# B&R Automation Studio project MotionTestBenchMaster (part 32)

```iecst
                               VAR_RNS_SEQ.Device.FSB201.ALR := FALSE;                                                 (* STEP: 93 FSB201*)
                               VAR_RNS_SEQ.Device.FSB201.WAIT_OFF := FALSE;
                               VAR_RNS_SEQ.Device.FSB201.WAIT_ON := FALSE;

                               VAR_RNS_SEQ.Device.FTB201.ALR_HighLimitEn := FALSE;                                     (* STEP: 93 FTB201*)
                               VAR_RNS_SEQ.Device.FTB201.ALR_HighLimitSP := 0;
                               VAR_RNS_SEQ.Device.FTB201.ALR_LowLimitEn := FALSE;
                               VAR_RNS_SEQ.Device.FTB201.ALR_LowLimitSP := 0;
                               VAR_RNS_SEQ.Device.FTB201.SP := 0;
                               VAR_RNS_SEQ.Device.FTB201.CMP := 0;
                               VAR_RNS_SEQ.Device.FTB201.MinDev := 0;
                               VAR_RNS_SEQ.Device.FTB201.MaxDev := 0;

                               VAR_RNS_SEQ.Device.FTB202.ALR_HighLimitEn := FALSE;                                     (* STEP: 93 FTB202*)
                               VAR_RNS_SEQ.Device.FTB202.ALR_HighLimitSP := 0;
                               VAR_RNS_SEQ.Device.FTB202.ALR_LowLimitEn := FALSE;
                               VAR_RNS_SEQ.Device.FTB202.ALR_LowLimitSP := 0;
                               VAR_RNS_SEQ.Device.FTB202.SP := 0;
                               VAR_RNS_SEQ.Device.FTB202.CMP := 0;
                               VAR_RNS_SEQ.Device.FTB202.MinDev := 0;
                               VAR_RNS_SEQ.Device.FTB202.MaxDev := 0;

                               VAR_RNS_SEQ.Device.PTB220.ALR_HighLimitEn := FALSE;                                     (* STEP: 93 PTB220*)
                               VAR_RNS_SEQ.Device.PTB220.ALR_HighLimitSP := 0;
                               VAR_RNS_SEQ.Device.PTB220.ALR_LowLimitEn := FALSE;
                               VAR_RNS_SEQ.Device.PTB220.ALR_LowLimitSP := 0;
                               VAR_RNS_SEQ.Device.PTB220.SP := 0;
                               VAR_RNS_SEQ.Device.PTB220.CMP := 0;
                               VAR_RNS_SEQ.Device.PTB220.MinDev := 0;
                               VAR_RNS_SEQ.Device.PTB220.MaxDev := 0;

                               VAR_RNS_SEQ.Device.PTB270.ALR_HighLimitEn := FALSE;                                     (* STEP: 93 PTB270*)
                               VAR_RNS_SEQ.Device.PTB270.ALR_HighLimitSP := 0;
                               VAR_RNS_SEQ.Device.PTB270.ALR_LowLimitEn := FALSE;
                               VAR_RNS_SEQ.Device.PTB270.ALR_LowLimitSP := 0;
                               VAR_RNS_SEQ.Device.PTB270.SP := 0;
                               VAR_RNS_SEQ.Device.PTB270.CMP := 0;
                               VAR_RNS_SEQ.Device.PTB270.MinDev := 0;
                               VAR_RNS_SEQ.Device.PTB270.MaxDev := 0;

                               VAR_RNS_SEQ.Device.LTB202.ALR_HighLimitEn := FALSE;                                     (* STEP: 93 LTB202*)
                               VAR_RNS_SEQ.Device.LTB202.ALR_HighLimitSP := 0;
                               VAR_RNS_SEQ.Device.LTB202.ALR_LowLimitEn := FALSE;
                               VAR_RNS_SEQ.Device.LTB202.ALR_LowLimitSP := 0;
                               VAR_RNS_SEQ.Device.LTB202.SP := 0;
                               VAR_RNS_SEQ.Device.LTB202.CMP := 0;
                               VAR_RNS_SEQ.Device.LTB202.MinDev := 0;
                               VAR_RNS_SEQ.Device.LTB202.MaxDev := 0;

                               VAR_RNS_SEQ.Device.PTB290.ALR_HighLimitEn := FALSE;                                     (* STEP: 93 PTB290*)
                               VAR_RNS_SEQ.Device.PTB290.ALR_HighLimitSP := 0;
                               VAR_RNS_SEQ.Device.PTB290.ALR_LowLimitEn := FALSE;
                               VAR_RNS_SEQ.Device.PTB290.ALR_LowLimitSP := 0;
                               VAR_RNS_SEQ.Device.PTB290.SP := 0;
                               VAR_RNS_SEQ.Device.PTB290.CMP := 0;
                               VAR_RNS_SEQ.Device.PTB290.MinDev := 0;
                               VAR_RNS_SEQ.Device.PTB290.MaxDev := 0;

                               VAR_RNS_SEQ.Mem.ContainersStop := TRUE;                                                 (* STEP: 93 *)
                               VAR_RNS_SEQ.Mem.ControlInsercion := FALSE;                                              (* STEP: 93 *)
                               VAR_RNS_SEQ.Mem.ControlContinous := FALSE;                                              (* STEP: 93 *)
                               VAR_RNS_SEQ.Mem.PBAbortEnable := TRUE;                                                  (* STEP: 93 PB Abort Sequence Enable*)
                               VAR_RNS_SEQ.Mem.PBStopEnable := TRUE;                                                   (* STEP: 93 PB Stop Sequence Enable*)
                               VAR_RNS_SEQ.Mem.PBStartEnable := FALSE;                                                 (* STEP: 93 PB Start Sequence Enable*)
                               VAR_RNS_SEQ.Mem.ByPassed := TRUE;                                                       (* STEP: 93 *)
                               VAR_RNS_SEQ.Mem.InsercionDevice := FALSE;                                               (* STEP: 93 *)
                               VAR_RNS_SEQ.Mem.AirTreatmentControl := FALSE;                                           (* STEP: 93 *)
                               VAR_RNS_SEQ.Mem.WaterTreatmentControl := FALSE;                                         (* STEP: 93 *)
                               VAR_RNS_SEQ.Mem.SpeedReductionControl := FALSE;                                         (* STEP: 93 *)
                               VAR_RNS_SEQ.Mem.ByPassRequest := FALSE;                                                 (* STEP: 93 *)
                               VAR_RNS_SEQ.Mem.CopAfterCipRequest := FALSE;                                            (* STEP: 93 *)
                               VAR_RNS_SEQ.Mem.NoBoNoSprayInsercion := FALSE;                                          (* STEP: 93 *)

                               VAR_RNS_SEQ.ITC.WTT_ProductRequest := FALSE;                                            (* STEP: 93 *)
                               VAR_RNS_SEQ.ITC.WTT_ProductionRunning := FALSE;                                         (* STEP: 93 *)

                       94: (* BYPASSED - Rinser Inserted  *)

                               VAR_RNS_SEQ.Device.AVB224.AutoCnd := FALSE;                                             (* STEP: 94 AVB224*)
                               VAR_RNS_SEQ.Device.AVB224.EnableCnd := FALSE;
                               VAR_RNS_SEQ.Device.AVB228.AutoCnd := FALSE;                                             (* STEP: 94 AVB228*)
                               VAR_RNS_SEQ.Device.AVB228.EnableCnd := FALSE;
                               VAR_RNS_SEQ.Device.AVB234.AutoCnd := FALSE;                                             (* STEP: 94 AVB234*)
                               VAR_RNS_SEQ.Device.AVB234.EnableCnd := FALSE;
                               VAR_RNS_SEQ.Device.AVB261.AutoCnd := FALSE;                                             (* STEP: 94 AVB261*)
                               VAR_RNS_SEQ.Device.AVB261.EnableCnd := FALSE;
                               VAR_RNS_SEQ.Device.AVB264.AutoCnd := FALSE;                                             (* STEP: 94 AVB264*)
                               VAR_RNS_SEQ.Device.AVB264.EnableCnd := FALSE;
                               VAR_RNS_SEQ.Device.AVB265.AutoCnd := FALSE;                                             (* STEP: 94 AVB265*)
                               VAR_RNS_SEQ.Device.AVB265.EnableCnd := FALSE;
                               VAR_RNS_SEQ.Device.AVB266.AutoCnd := FALSE;                                             (* STEP: 94 AVB266*)
                               VAR_RNS_SEQ.Device.AVB266.EnableCnd := FALSE;
                               VAR_RNS_SEQ.Device.AVB267.AutoCnd := FALSE;                                             (* STEP: 94 AVB267*)
                               VAR_RNS_SEQ.Device.AVB267.EnableCnd := FALSE;
                               VAR_RNS_SEQ.Device.AVB268.AutoCnd := FALSE;                                             (* STEP: 94 AVB268*)
                               VAR_RNS_SEQ.Device.AVB268.EnableCnd := FALSE;
                               VAR_RNS_SEQ.Device.AVB273.AutoCnd := FALSE;                                             (* STEP: 94 AVB273*)
                               VAR_RNS_SEQ.Device.AVB273.EnableCnd := FALSE;
                               VAR_RNS_SEQ.Device.AVB294.AutoCnd := FALSE;                                             (* STEP: 94 AVB294*)
                               VAR_RNS_SEQ.Device.AVB294.EnableCnd := FALSE;

                               VAR_RNS_SEQ.Device.PPB209_PID.PID_Enable := FALSE;                                      (* STEP: 94 PPB209*)
                               VAR_RNS_SEQ.Device.PPB209_PID.PID_Mode := FALSE;
                               VAR_RNS_SEQ.Device.PPB209_PID.Auto_SP_Value := 0;
                               VAR_RNS_SEQ.Device.PPB209_PID.FIX_Value := 0;

                               VAR_RNS_SEQ.Device.RVB202_PID.PID_Enable := FALSE;                                      (* STEP: 94 *)
                               VAR_RNS_SEQ.Device.RVB202_PID.PID_Mode := FALSE;
                               VAR_RNS_SEQ.Device.RVB202_PID.Auto_SP_Value := 0;
                               VAR_RNS_SEQ.Device.RVB202_PID.FIX_Value := 0;

                               VAR_RNS_SEQ.Device.FSB220.ALR := FALSE;                                                 (* STEP: 94 FSB220*)
                               VAR_RNS_SEQ.Device.FSB220.WAIT_OFF := FALSE;
                               VAR_RNS_SEQ.Device.FSB220.WAIT_ON := FALSE;

                               VAR_RNS_SEQ.Device.LSB209.ALR := FALSE;                                                 (* STEP: 94 LSB209*)
                               VAR_RNS_SEQ.Device.LSB209.WAIT_OFF := FALSE;
                               VAR_RNS_SEQ.Device.LSB209.WAIT_ON := FALSE;

                               VAR_RNS_SEQ.Device.LSB210.ALR := FALSE;                                                 (* STEP: 94 LSB210*)
                               VAR_RNS_SEQ.Device.LSB210.WAIT_OFF := FALSE;
                               VAR_RNS_SEQ.Device.LSB210.WAIT_ON := FALSE;

                               VAR_RNS_SEQ.Device.LSB299.ALR := FALSE;                                                 (* STEP: 94 *)
                               VAR_RNS_SEQ.Device.LSB299.WAIT_OFF := FALSE;
                               VAR_RNS_SEQ.Device.LSB299.WAIT_ON := FALSE;

                               VAR_RNS_SEQ.Device.FSB201.ALR := FALSE;                                                 (* STEP: 94 FSB201*)
                               VAR_RNS_SEQ.Device.FSB201.WAIT_OFF := FALSE;
                               VAR_RNS_SEQ.Device.FSB201.WAIT_ON := FALSE;

                               VAR_RNS_SEQ.Device.FTB201.ALR_HighLimitEn := FALSE;                                     (* STEP: 94 FTB201*)
                               VAR_RNS_SEQ.Device.FTB201.ALR_HighLimitSP := 0;
                               VAR_RNS_SEQ.Device.FTB201.ALR_LowLimitEn := FALSE;
                               VAR_RNS_SEQ.Device.FTB201.ALR_LowLimitSP := 0;
                               VAR_RNS_SEQ.Device.FTB201.SP := 0;
                               VAR_RNS_SEQ.Device.FTB201.CMP := 0;
                               VAR_RNS_SEQ.Device.FTB201.MinDev := 0;
                               VAR_RNS_SEQ.Device.FTB201.MaxDev := 0;

                               VAR_RNS_SEQ.Device.FTB202.ALR_HighLimitEn := FALSE;                                     (* STEP: 94 FTB202*)
                               VAR_RNS_SEQ.Device.FTB202.ALR_HighLimitSP := 0;
                               VAR_RNS_SEQ.Device.FTB202.ALR_LowLimitEn := FALSE;
                               VAR_RNS_SEQ.Device.FTB202.ALR_LowLimitSP := 0;
                               VAR_RNS_SEQ.Device.FTB202.SP := 0;
                               VAR_RNS_SEQ.Device.FTB202.CMP := 0;
                               VAR_RNS_SEQ.Device.FTB202.MinDev := 0;
                               VAR_RNS_SEQ.Device.FTB202.MaxDev := 0;

                               VAR_RNS_SEQ.Device.PTB220.ALR_HighLimitEn := FALSE;                                     (* STEP: 94 PTB220*)
                               VAR_RNS_SEQ.Device.PTB220.ALR_HighLimitSP := 0;
                               VAR_RNS_SEQ.Device.PTB220.ALR_LowLimitEn := FALSE;
                               VAR_RNS_SEQ.Device.PTB220.ALR_LowLimitSP := 0;
                               VAR_RNS_SEQ.Device.PTB220.SP := 0;
                               VAR_RNS_SEQ.Device.PTB220.CMP := 0;
                               VAR_RNS_SEQ.Device.PTB220.MinDev := 0;
                               VAR_RNS_SEQ.Device.PTB220.MaxDev := 0;

                               VAR_RNS_SEQ.Device.PTB270.ALR_HighLimitEn := FALSE;                                     (* STEP: 94 PTB270*)
                               VAR_RNS_SEQ.Device.PTB270.ALR_HighLimitSP := 0;
                               VAR_RNS_SEQ.Device.PTB270.ALR_LowLimitEn := FALSE;
                               VAR_RNS_SEQ.Device.PTB270.ALR_LowLimitSP := 0;
                               VAR_RNS_SEQ.Device.PTB270.SP := 0;
                               VAR_RNS_SEQ.Device.PTB270.CMP := 0;
                               VAR_RNS_SEQ.Device.PTB270.MinDev := 0;
                               VAR_RNS_SEQ.Device.PTB270.MaxDev := 0;

                               VAR_RNS_SEQ.Device.LTB202.ALR_HighLimitEn := FALSE;                                     (* STEP: 94 LTB202*)
                               VAR_RNS_SEQ.Device.LTB202.ALR_HighLimitSP := 0;
                               VAR_RNS_SEQ.Device.LTB202.ALR_LowLimitEn := FALSE;
                               VAR_RNS_SEQ.Device.LTB202.ALR_LowLimitSP := 0;
                               VAR_RNS_SEQ.Device.LTB202.SP := 0;
                               VAR_RNS_SEQ.Device.LTB202.CMP := 0;
                               VAR_RNS_SEQ.Device.LTB202.MinDev := 0;
                               VAR_RNS_SEQ.Device.LTB202.MaxDev := 0;

                               VAR_RNS_SEQ.Device.PTB290.ALR_HighLimitEn := FALSE;                                     (* STEP: 94 PTB290*)
                               VAR_RNS_SEQ.Device.PTB290.ALR_HighLimitSP := 0;
                               VAR_RNS_SEQ.Device.PTB290.ALR_LowLimitEn := FALSE;
                               VAR_RNS_SEQ.Device.PTB290.ALR_LowLimitSP := 0;
                               VAR_RNS_SEQ.Device.PTB290.SP := 0;
                               VAR_RNS_SEQ.Device.PTB290.CMP := 0;
                               VAR_RNS_SEQ.Device.PTB290.MinDev := 0;
                               VAR_RNS_SEQ.Device.PTB290.MaxDev := 0;

                               VAR_RNS_SEQ.Mem.ContainersStop := TRUE;                                                 (* STEP: 94 *)
                               VAR_RNS_SEQ.Mem.ControlInsercion := FALSE;                                              (* STEP: 94 *)
                               VAR_RNS_SEQ.Mem.ControlContinous := FALSE;                                              (* STEP: 94 *)
                               VAR_RNS_SEQ.Mem.PBAbortEnable := TRUE;                                                  (* STEP: 94 PB Abort Sequence Enable*)
                               VAR_RNS_SEQ.Mem.PBStopEnable := TRUE;                                                   (* STEP: 94 PB Stop Sequence Enable*)
                               VAR_RNS_SEQ.Mem.PBStartEnable := FALSE;                                                 (* STEP: 94 PB Start Sequence Enable*)
                               VAR_RNS_SEQ.Mem.ByPassed := FALSE;                                                      (* STEP: 94 *)
                               VAR_RNS_SEQ.Mem.InsercionDevice := FALSE;                                               (* STEP: 94 *)
                               VAR_RNS_SEQ.Mem.AirTreatmentControl := FALSE;                                           (* STEP: 94 *)
                               VAR_RNS_SEQ.Mem.WaterTreatmentControl := FALSE;                                         (* STEP: 94 *)
                               VAR_RNS_SEQ.Mem.SpeedReductionControl := FALSE;                                         (* STEP: 94 *)
                               VAR_RNS_SEQ.Mem.ByPassRequest := TRUE;                                                  (* STEP: 94 *)
                               VAR_RNS_SEQ.Mem.CopAfterCipRequest := FALSE;                                            (* STEP: 94 *)
                               VAR_RNS_SEQ.Mem.NoBoNoSprayInsercion := FALSE;                                          (* STEP: 94 *)

                               VAR_RNS_SEQ.ITC.WTT_ProductRequest := FALSE;                                            (* STEP: 94 *)
                               VAR_RNS_SEQ.ITC.WTT_ProductionRunning := FALSE;                                         (* STEP: 94 *)

                       95..100: (* Spare Steps *)

               ELSE
                               RNS_StepStop;
               END_CASE
END_ACTION
```

#### RNS_StepStatus.st
```iecst
ACTION RNS_StepStatus:
	//MODE
	VAR_RNS_ModeWait					:= VAR_RNS_SeqPermanent.SeqActualStep = 0;
	VAR_RNS_ModeProduction				:= VAR_RNS_SeqPermanent.SeqMode1.0;
	VAR_RNS_ModeCip						:= VAR_RNS_SeqPermanent.SeqMode1.1;
	VAR_RNS_ModeDrain					:= VAR_RNS_SeqPermanent.SeqMode1.3;
	VAR_RNS_ModeCop						:= VAR_RNS_SeqPermanent.SeqMode1.4;
	VAR_RNS_ModeControl					:= VAR_RNS_SeqPermanent.SeqMode1.5 OR VAR_RNS_SeqPermanent.SeqMode2.1;//V4.A.A.1.7.0
	VAR_RNS_ModeBypass					:= VAR_RNS_SeqPermanent.SeqMode1.6;//V4.A.A.1.7.0
	VAR_RNS_ModeDeEnergization 			:= VAR_RNS_SeqPermanent.SeqMode1.14;
	VAR_RNS_ModeFiltersSterilization 	:= VAR_RNS_SeqPermanent.SeqMode1.15;

	VAR_RNS_MemProdDrain				:= VAR_RNS_SeqPermanent.SeqMode2.0;//V4.A.A.1.7.0
	VAR_RNS_MemProdControl				:= VAR_RNS_SeqPermanent.SeqMode2.1;//V4.A.A.1.7.0
	VAR_RNS_MemRinserByPassed			:= VAR_RNS_SeqPermanent.SeqMode2.2;//V4.A.A.1.7.0
	VAR_RNS_MemRinserInserted			:= VAR_RNS_SeqPermanent.SeqMode2.3;//V4.A.A.1.7.0
	VAR_RNS_ModeWaitOperator			:= FALSE;

	//STEP PRODUCTION
	VAR_RNS_StepProdStartUp				:= VAR_RNS_SeqActualStep >= 10 AND VAR_RNS_SeqActualStep <= 19;
	//VAR_RNS_StepProdStartUpLampCtrl	:= VAR_RNS_SeqActualStep >= 10 AND VAR_RNS_SeqActualStep <= 12;
	//VAR_RNS_StepProdStartUpLampFault	:= VAR_RNS_SeqActualStep = 13;
	VAR_RNS_StepProdProducing			:= VAR_RNS_SeqActualStep >= 20 AND VAR_RNS_SeqActualStep <= 29;
	//VAR_RNS_StepProdSprayRequest		:= VAR_RNS_SeqActualStep >= 22 AND VAR_RNS_SeqActualStep <= 28;
	VAR_RNS_StepProdStopped				:= VAR_RNS_SeqActualStep = 31;
	VAR_RNS_StepProdAborted				:= VAR_RNS_SeqActualStep = 0;

	//STEP CIP
	VAR_RNS_StepCipCleaning			:= VAR_RNS_SeqActualStep = 41;
	VAR_RNS_StepCipEnded			:= VAR_RNS_SeqActualStep = 48;

	//STEP DRAIN
	VAR_RNS_StepDrainStopped			:= VAR_RNS_SeqActualStep = 54;
	VAR_RNS_StepDrainAborted			:= VAR_RNS_SeqActualStep = 0;

	//STEP CONTROL
	VAR_RNS_StepControl					:= VAR_RNS_SeqActualStep >= 70 AND VAR_RNS_SeqActualStep <= 80;//V4.A.A.1.7.0
	VAR_RNS_StepControlDone				:= VAR_RNS_SeqActualStep = 81;
	VAR_RNS_StepControlStopped			:= VAR_RNS_SeqActualStep = 80;
	VAR_RNS_StepControlAborted			:= VAR_RNS_SeqActualStep = 0 OR VAR_RNS_SeqActualStep = 80;

	IF VAR_RNS_StepControlDone THEN
		VAR_RNS_StepCtrlCipDone := TRUE;
	END_IF

	IF VAR_RNS_SeqActualStep = 55 OR VAR_RNS_SeqActualStep = 48 OR VAR_RNS_SeqActualStep = 0 THEN
		VAR_RNS_StepCtrlCipDone := FALSE;
	END_IF

	//STEP CIP
	VAR_RNS_StepCipCleaning		:= VAR_RNS_SeqActualStep = 41;
	VAR_RNS_StepCipStopped		:= VAR_RNS_SeqActualStep = 0 OR VAR_RNS_SeqActualStep = 49 OR VAR_RNS_SeqActualStep = 101;//vrma
	VAR_RNS_StepCipAborted		:= VAR_RNS_SeqActualStep = 0 OR VAR_RNS_SeqActualStep = 49;

	//STEP BYPASS
	VAR_RNS_StepByPassed					:= VAR_RNS_SeqActualStep >= 90 AND VAR_RNS_SeqActualStep <= 95;//V4.A.A.1.7.0
	VAR_RNS_StepBypassAborted				:= VAR_RNS_SeqActualStep = 0;

	IF FB_RNS_SEQ.OUT_StepActual = 91 THEN
		VAR_RNS_BypassCommand := TRUE;
	ELSIF FB_RNS_SEQ.OUT_StepActual = 94 THEN
		VAR_RNS_BypassCommand := FALSE;
	ELSE
	END_IF

	IF RNS.DataOut.ByPassed THEN
		VAR_RNS_SeqPermanent.SeqMode2.2 := TRUE;
		VAR_RNS_SeqPermanent.SeqMode2.3 := FALSE;
	ELSE
		VAR_RNS_SeqPermanent.SeqMode2.3 := TRUE;
		VAR_RNS_SeqPermanent.SeqMode2.2 := FALSE;
	END_IF

END_ACTION
```

#### RNS_StepStop.st
```iecst
ACTION RNS_StepStop:

		VAR_RNS_SEQ.Device.AVB224.AutoCnd := TRUE;                                              (* STEP: 101 *)
		VAR_RNS_SEQ.Device.AVB224.EnableCnd := TRUE;
		VAR_RNS_SEQ.Device.AVB228.AutoCnd := FALSE;                                             (* STEP: 101 *)
		VAR_RNS_SEQ.Device.AVB228.EnableCnd := FALSE;
		VAR_RNS_SEQ.Device.AVB261.AutoCnd := FALSE;                                              (* STEP: 101 *)
		VAR_RNS_SEQ.Device.AVB261.EnableCnd := FALSE;
		VAR_RNS_SEQ.Device.AVB267.AutoCnd := FALSE;                                             (* STEP: 101 *)
		VAR_RNS_SEQ.Device.AVB267.EnableCnd := FALSE;
		VAR_RNS_SEQ.Device.AVB268.AutoCnd := FALSE;                                             (* STEP: 101 *)
		VAR_RNS_SEQ.Device.AVB268.EnableCnd := FALSE;
		VAR_RNS_SEQ.Device.AVB273.AutoCnd := FALSE;                                             (* STEP: 101 *)
		VAR_RNS_SEQ.Device.AVB273.EnableCnd := FALSE;

	VAR_RNS_SEQ.Device.PPB209_PID.PID_Enable := FALSE;                                      (* STEP: 101 *)
	VAR_RNS_SEQ.Device.PPB209_PID.PID_Mode := FALSE;
	VAR_RNS_SEQ.Device.PPB209_PID.Auto_SP_Value := 0;
	VAR_RNS_SEQ.Device.PPB209_PID.FIX_Value := 0;

	VAR_RNS_SEQ.Device.LSB209.ALR := FALSE;                                                (* STEP: 101 *)
	VAR_RNS_SEQ.Device.LSB209.WAIT_OFF := FALSE;
	VAR_RNS_SEQ.Device.LSB209.WAIT_ON := FALSE;

	VAR_RNS_SEQ.Device.LSB299.ALR := FALSE;                                                (* STEP: 101 *)
	VAR_RNS_SEQ.Device.LSB299.WAIT_OFF := FALSE;
	VAR_RNS_SEQ.Device.LSB299.WAIT_ON := FALSE;

	VAR_RNS_SEQ.Device.LSB210.ALR := FALSE;                                                (* STEP: 101 *)
	VAR_RNS_SEQ.Device.LSB210.WAIT_OFF := FALSE;
	VAR_RNS_SEQ.Device.LSB210.WAIT_ON := FALSE;

	VAR_RNS_SEQ.Device.FSB201.ALR := FALSE;                                                 (* STEP: 101 *)
	VAR_RNS_SEQ.Device.FSB201.WAIT_OFF := FALSE;
	VAR_RNS_SEQ.Device.FSB201.WAIT_ON := FALSE;

	VAR_RNS_SEQ.Device.FSB220.ALR := FALSE;                                                 (* STEP: 101 *)
	VAR_RNS_SEQ.Device.FSB220.WAIT_OFF := FALSE;
	VAR_RNS_SEQ.Device.FSB220.WAIT_ON := FALSE;

	VAR_RNS_SEQ.Device.FTB201.ALR_HighLimitEn := FALSE;                                     (* STEP: 101 *)
	VAR_RNS_SEQ.Device.FTB201.ALR_HighLimitSP := 0;
	VAR_RNS_SEQ.Device.FTB201.ALR_LowLimitEn := FALSE;
	VAR_RNS_SEQ.Device.FTB201.ALR_LowLimitSP := 0;
	VAR_RNS_SEQ.Device.FTB201.SP := 0;
	VAR_RNS_SEQ.Device.FTB201.CMP := 0;
	VAR_RNS_SEQ.Device.FTB201.MinDev := 0;
	VAR_RNS_SEQ.Device.FTB201.MaxDev := 0;

	VAR_RNS_SEQ.Device.FTB202.ALR_HighLimitEn := FALSE;                                     (* STEP: 101 *)
	VAR_RNS_SEQ.Device.FTB201.ALR_HighLimitSP := 0;
	VAR_RNS_SEQ.Device.FTB202.ALR_LowLimitEn := FALSE;
	VAR_RNS_SEQ.Device.FTB202.ALR_LowLimitSP := 0;
	VAR_RNS_SEQ.Device.FTB202.SP := 0;
	VAR_RNS_SEQ.Device.FTB202.CMP := 0;
	VAR_RNS_SEQ.Device.FTB202.MinDev := 0;
	VAR_RNS_SEQ.Device.FTB202.MaxDev := 0;

	VAR_RNS_SEQ.Device.PTB220.ALR_HighLimitEn := FALSE;                                     (* STEP: 101 *)
	VAR_RNS_SEQ.Device.PTB220.ALR_HighLimitSP := 0;
	VAR_RNS_SEQ.Device.PTB220.ALR_LowLimitEn := FALSE;
	VAR_RNS_SEQ.Device.PTB220.ALR_LowLimitSP := 0;
	VAR_RNS_SEQ.Device.PTB220.SP := 0;
	VAR_RNS_SEQ.Device.PTB220.CMP := 0;
	VAR_RNS_SEQ.Device.PTB220.MinDev := 0;
	VAR_RNS_SEQ.Device.PTB220.MaxDev := 0;

	VAR_RNS_SEQ.Device.PTB270.ALR_HighLimitEn := FALSE;                                     (* STEP: 101 *)
	VAR_RNS_SEQ.Device.PTB270.ALR_HighLimitSP := 0;
	VAR_RNS_SEQ.Device.PTB270.ALR_LowLimitEn := FALSE;
	VAR_RNS_SEQ.Device.PTB270.ALR_LowLimitSP := 0;
	VAR_RNS_SEQ.Device.PTB270.SP := 0;
	VAR_RNS_SEQ.Device.PTB270.CMP := 0;
	VAR_RNS_SEQ.Device.PTB270.MinDev := 0;
	VAR_RNS_SEQ.Device.PTB270.MaxDev := 0;

	VAR_RNS_SEQ.Mem.ContainersStop := TRUE;                                               	(* STEP: 101 *)
END_ACTION
```

#### RNS_ValvesLogic.st
```iecst
ACTION RNS_ValvesLogic:
	TOF_StatusMachineRunning.IN	:= SEL(MC_InputOutput.Network.Machine.Status.MultiModalityActive, MC_InputOutput.Network.Machine.Status.MachineRunning, MC_InputOutput.Network.Filler.Status.ModuleRunning);
	TOF_StatusMachineRunning.PT := t#10s;
	TOF_StatusMachineRunning();

	VAR_RNS_ValveEnable 	:= OPS.DataOut.EmergencyOk;
	VAR_RNS_ValveEnableCip 	:= OPS.DataOut.EmergencyOk AND OPS.DataOut.DoorsOk;

	//AVB224 RINSER DISCHARGE
	AVB[224].IN_Enable		:= VAR_RNS_ValveEnable;
	AVB[224].IN_AutoCnd		:= VAR_RNS_SEQ.Device.AVB224.AutoCnd;
	AVB[224].IN_EnableCnd	:= VAR_RNS_SEQ.Device.AVB224.EnableCnd;
	AVB[224].IN_Cnd 		:= NOT VAR_RNS_WaterTreatment;
	AVB[224].IN_ManEn		:= TRUE;
	AVB[224].IN_MaskEn		:= TRUE;

	//AVB228 RINSER DISCHARGE
	AVB[228].IN_Enable		:= VAR_RNS_ValveEnable;
	AVB[228].IN_AutoCnd		:= VAR_RNS_SEQ.Device.AVB228.AutoCnd OR TOF_StatusMachineRunning.Q;//vrma
	AVB[228].IN_EnableCnd	:= VAR_RNS_SEQ.Device.AVB228.EnableCnd;
	AVB[228].IN_Cnd 		:= MNM.DataOut.MachineRunning;//vrma
	AVB[228].IN_ManEn		:= TRUE;
	AVB[228].IN_MaskEn		:= TRUE;

	//AVB234 TWISTER DISCHARGE
	AVB[234].IN_Enable      := VAR_RNS_ValveEnable;
	AVB[234].IN_AutoCnd     := VAR_RNS_SEQ.Device.AVB234.AutoCnd;//vrma
	AVB[234].IN_EnableCnd   := VAR_RNS_SEQ.Device.AVB234.EnableCnd;
	AVB[234].IN_Cnd         := FALSE;
	AVB[234].IN_ManEn       := TRUE;
	AVB[234].IN_MaskEn      := TRUE;

	//AVB261 H2O RINSING VALVE
	AVB[261].IN_Enable		:= VAR_RNS_ValveEnable;
	AVB[261].IN_AutoCnd		:= VAR_RNS_SEQ.Device.AVB261.AutoCnd;
	AVB[261].IN_EnableCnd	:= VAR_RNS_SEQ.Device.AVB261.EnableCnd;
	AVB[261].IN_Cnd 		:= MNM.DataOut.MachineRunning;//vrma
	AVB[261].IN_ManEn		:= TRUE;
	AVB[261].IN_MaskEn		:= TRUE;

	//AVB264 RINSING CIP VALVE //V4.A.A.1.7.0
	AVB[264].IN_Enable		:= VAR_RNS_ValveEnableCip AND (TNK.DataOut.ProdMode OR TNK.DataOut.Wait);
	AVB[264].IN_AutoCnd		:= VAR_RNS_SEQ.Device.AVB264.AutoCnd;
	AVB[264].IN_EnableCnd	:= VAR_RNS_SEQ.Device.AVB264.EnableCnd;
	AVB[264].IN_Cnd 		:= VAR_RNS_WaterTreatment AND NOT VAR_RNS_CleaningActive;
	AVB[264].IN_ManEn		:= TRUE;
	AVB[264].IN_MaskEn		:= TRUE;

	//AVB265 RINSING CIP VALVE //V4.A.A.1.7.0
	AVB[265].IN_Enable		:= VAR_RNS_ValveEnableCip;
	AVB[265].IN_AutoCnd		:= VAR_RNS_SEQ.Device.AVB265.AutoCnd;
	AVB[265].IN_EnableCnd	:= VAR_RNS_SEQ.Device.AVB265.EnableCnd;
	AVB[265].IN_Cnd 		:= VAR_RNS_WaterTreatment;
	AVB[265].IN_ManEn		:= TRUE;
	AVB[265].IN_MaskEn		:= TRUE;

	//AVB265 RINSING CIP VALVE //V4.A.A.1.7.0
	AVB[266].IN_Enable		:= VAR_RNS_ValveEnableCip;
	AVB[266].IN_AutoCnd		:= VAR_RNS_SEQ.Device.AVB266.AutoCnd OR TOF_StatusMachineRunning.Q;//vrma
	AVB[266].IN_EnableCnd	:= VAR_RNS_SEQ.Device.AVB266.EnableCnd;
	AVB[266].IN_Cnd 		:= FALSE;
	AVB[266].IN_ManEn		:= TRUE;
	AVB[266].IN_MaskEn		:= TRUE;

	//AVB267 CIP DRAIN v1.4
	AVB[267].IN_Enable		:= VAR_RNS_ValveEnable;
	AVB[267].IN_AutoCnd		:= VAR_RNS_SEQ.Device.AVB267.AutoCnd;
	AVB[267].IN_EnableCnd	:= VAR_RNS_SEQ.Device.AVB267.EnableCnd;
	AVB[267].IN_Cnd 		:= FALSE;
	AVB[267].IN_ManEn		:= TRUE;
	AVB[267].IN_MaskEn		:= TRUE;

	//AVB268 COP/CIP DRAIN v1.4
	AVB[268].IN_Enable		:= VAR_RNS_ValveEnable;
	AVB[268].IN_AutoCnd		:= VAR_RNS_SEQ.Device.AVB268.AutoCnd;
	AVB[268].IN_EnableCnd	:= VAR_RNS_SEQ.Device.AVB268.EnableCnd;
	AVB[268].IN_Cnd 		:= FALSE;
	AVB[268].IN_ManEn		:= TRUE;
	AVB[268].IN_MaskEn		:= TRUE;

	//AVB273 AIR RINSING VALVE
	AVB[273].IN_Enable		:= VAR_RNS_ValveEnable;
	AVB[273].IN_AutoCnd		:= VAR_RNS_SEQ.Device.AVB273.AutoCnd;
	AVB[273].IN_EnableCnd	:= VAR_RNS_SEQ.Device.AVB273.EnableCnd;
	AVB[273].IN_Cnd 		:= VAR_RNS_AirTreatment;
	AVB[273].IN_ManEn		:= TRUE;
	AVB[273].IN_MaskEn		:= TRUE;

	//DYNAMIC COMMAND
	TMR_TON_FlipWait.IN	:= VAR_RNS_StepCipCleaning AND NOT TMR_TOF_FlipWork.Q AND NOT (LTB[202].OUT_ActValue >70.0);
	TMR_TON_FlipWait.PT	:= REAL_TO_TIME(60.0*1000); //[ms]*1000
	TMR_TON_FlipWait();

	TMR_TOF_FlipWork.IN := TMR_TON_FlipWait.Q;
	TMR_TOF_FlipWork.PT := REAL_TO_TIME(4.0*1000); //[ms]*1000
	TMR_TOF_FlipWork();

	//AVB294
	IF VAR_RNS_ModeProduction THEN//vrma
		IF LTB[202].OUT_ActValue >70.0 THEN
			AVB[294].IN_AutoCnd := FALSE;
		ELSIF LTB[202].OUT_ActValue < 20.0 THEN
			AVB[294].IN_AutoCnd	:= TRUE;
		END_IF
	ELSIF VAR_RNS_ModeCip THEN //FACCIAMO FLIP
		AVB[294].IN_AutoCnd := TMR_TOF_FlipWork.Q;
	ELSE
		AVB[294].IN_AutoCnd := FALSE;
	END_IF

	AVB[294].IN_Enable		:= VAR_RNS_ValveEnable;
	AVB[294].IN_AutoCnd		:= FALSE; // leo AVB[294].IN_AutoCnd;
	AVB[294].IN_EnableCnd	:= FALSE;
	AVB[294].IN_Cnd 		:= VAR_RNS_AirTreatment;
	AVB[294].IN_ManEn		:= TRUE;
	AVB[294].IN_MaskEn		:= TRUE;

END_ACTION
```

#### RNS_ValvesFB.st
```iecst
ACTION RNS_ValvesFB:
//AVB224 RINSER DISCHARGE
	AVB[224](
	IN_ConfigPresent 	:= AVB[224].IN_ConfigPresent,
	IN_Enable 			:= AVB[224].IN_Enable,
	IN_AutoCnd 			:= AVB[224].IN_AutoCnd,
	IN_EnableCnd 		:= AVB[224].IN_EnableCnd,
	IN_Cnd 				:= AVB[224].IN_Cnd,
	IN_FlipEnable 		:= FALSE,
	IN_FlipRequest		:= FALSE,
	IN_FlipTime 		:= T#500ms,
	IN_Reset 			:= VAR_RNS_PBResetEp,
	IN_HMIAutoForce 	:= NOT HMI_SS2P[SS2P_HMI_DeviceEnable].ON,
	IN_ManEn 			:= AVB[224].IN_ManEn,
	IN_MaskEn 			:= AVB[224].IN_MaskEn,
	IO 					:= IO_AVB[224],
	HMI 				:= HMI_AVB[224]
	);

	//AVB228 H2O EXTERNAL RINSING VALVE
	AVB[228](
	IN_ConfigPresent 	:= AVB[228].IN_ConfigPresent,
	IN_Enable 			:= AVB[228].IN_Enable,
	IN_AutoCnd 			:= AVB[228].IN_AutoCnd,
	IN_EnableCnd 		:= AVB[228].IN_EnableCnd,
	IN_Cnd 				:= AVB[228].IN_Cnd,
	IN_FlipEnable 		:= FALSE,
	IN_FlipRequest		:= FALSE,
	IN_FlipTime 		:= T#500ms,
	IN_Reset 			:= VAR_RNS_PBResetEp,
	IN_HMIAutoForce 	:= NOT HMI_SS2P[SS2P_HMI_DeviceEnable].ON,
	IN_ManEn 			:= AVB[228].IN_ManEn,
	IN_MaskEn 			:= AVB[228].IN_MaskEn,
	IO 					:= IO_AVB[228],
	HMI 				:= HMI_AVB[228]
	);

	//AVB234 TWIST COOLING DRAIN
	AVB[234](//VRMA
	IN_ConfigPresent          := AVB[234].IN_ConfigPresent,
	IN_Enable                 := AVB[234].IN_Enable,
	IN_AutoCnd                := AVB[234].IN_AutoCnd,
	IN_EnableCnd              := AVB[234].IN_EnableCnd,
	IN_Cnd                    := AVB[234].IN_Cnd,
	IN_FlipEnable             := FALSE,
	IN_FlipRequest            := FALSE,
	IN_FlipTime               := T#500ms,
	IN_Reset                  := VAR_RNS_PBResetEp,
	IN_HMIAutoForce           := NOT HMI_SS2P[SS2P_HMI_DeviceEnable].ON,
	IN_ManEn                  := AVB[234].IN_ManEn,
	IN_MaskEn                 := AVB[234].IN_MaskEn,
	IO                        := IO_AVB[234],
	HMI                       := HMI_AVB[234]);

	//AVB261 H2O RINSING VALVE
	AVB[261](
	IN_ConfigPresent 	:= AVB[261].IN_ConfigPresent,
	IN_Enable 			:= AVB[261].IN_Enable,
	IN_AutoCnd 			:= AVB[261].IN_AutoCnd,
	IN_EnableCnd 		:= AVB[261].IN_EnableCnd,
	IN_Cnd 				:= AVB[261].IN_Cnd,
	IN_FlipEnable 		:= FALSE,
	IN_FlipRequest		:= FALSE,
	IN_FlipTime 		:= T#500ms,
	IN_Reset 			:= VAR_RNS_PBResetEp,
	IN_HMIAutoForce 	:= NOT HMI_SS2P[SS2P_HMI_DeviceEnable].ON,
	IN_ManEn 			:= AVB[261].IN_ManEn,
	IN_MaskEn 			:= AVB[261].IN_MaskEn,
	IO 					:= IO_AVB[261],
	HMI 				:= HMI_AVB[261]
	);

	//AVB264 RINSING CIP VALVE //V4.A.A.1.7.0
	AVB[264](
	IN_ConfigPresent 	:= AVB[264].IN_ConfigPresent,
	IN_Enable 			:= AVB[264].IN_Enable,
	IN_AutoCnd 			:= AVB[264].IN_AutoCnd,
	IN_EnableCnd 		:= AVB[264].IN_EnableCnd,
	IN_Cnd 				:= AVB[264].IN_Cnd,
	IN_FlipEnable 		:= FALSE,
	IN_FlipRequest		:= FALSE,
	IN_FlipTime 		:= T#500ms,
	IN_Reset 			:= VAR_RNS_PBResetEp,
	IN_HMIAutoForce 	:= NOT HMI_SS2P[SS2P_HMI_DeviceEnable].ON,
	IN_ManEn 			:= AVB[264].IN_ManEn,
	IN_MaskEn 			:= AVB[264].IN_MaskEn,
	IO 					:= IO_AVB[264],
	HMI 				:= HMI_AVB[264]
	);

	//AVB265 RINSING CIP VALVE //V4.A.A.1.7.0
	AVB[265](
	IN_ConfigPresent 	:= AVB[265].IN_ConfigPresent,
	IN_Enable 			:= AVB[265].IN_Enable,
	IN_AutoCnd 			:= AVB[265].IN_AutoCnd,
	IN_EnableCnd 		:= AVB[265].IN_EnableCnd,
	IN_Cnd 				:= AVB[265].IN_Cnd,
	IN_FlipEnable 		:= FALSE,
	IN_FlipRequest		:= FALSE,
	IN_FlipTime 		:= T#500ms,
	IN_Reset 			:= VAR_RNS_PBResetEp,
	IN_HMIAutoForce 	:= NOT HMI_SS2P[SS2P_HMI_DeviceEnable].ON,
	IN_ManEn 			:= AVB[265].IN_ManEn,
	IN_MaskEn 			:= AVB[265].IN_MaskEn,
	IO 					:= IO_AVB[265],
	HMI 				:= HMI_AVB[265]
	);

	//AVB266 RINSING CIP VALVE //V4.A.A.1.7.0
	AVB[266](
	IN_ConfigPresent 	:= AVB[266].IN_ConfigPresent,
	IN_Enable 			:= AVB[266].IN_Enable,
	IN_AutoCnd 			:= AVB[266].IN_AutoCnd,
	IN_EnableCnd 		:= AVB[266].IN_EnableCnd,
	IN_Cnd 				:= AVB[266].IN_Cnd,
	IN_FlipEnable 		:= FALSE,
	IN_FlipRequest		:= FALSE,
	IN_FlipTime 		:= T#500ms,
	IN_Reset 			:= VAR_RNS_PBResetEp,
	IN_HMIAutoForce 	:= NOT HMI_SS2P[SS2P_HMI_DeviceEnable].ON,
	IN_ManEn 			:= AVB[266].IN_ManEn,
	IN_MaskEn 			:= AVB[266].IN_MaskEn,
	IO 					:= IO_AVB[266],
	HMI 				:= HMI_AVB[266]
	);

	//AVB267 CIP To DRAIN v1.4
	AVB[267](
	IN_ConfigPresent 	:= AVB[267].IN_ConfigPresent,
	IN_Enable 			:= AVB[267].IN_Enable,
	IN_AutoCnd 			:= AVB[267].IN_AutoCnd,
	IN_EnableCnd 		:= AVB[267].IN_EnableCnd,
	IN_Cnd 				:= AVB[267].IN_Cnd,
	IN_FlipEnable 		:= FALSE,
	IN_FlipRequest		:= FALSE,
	IN_FlipTime 		:= T#500ms,
	IN_Reset 			:= VAR_RNS_PBResetEp,
	IN_HMIAutoForce 	:= NOT HMI_SS2P[SS2P_HMI_DeviceEnable].ON,
	IN_ManEn 			:= AVB[267].IN_ManEn,
	IN_MaskEn 			:= AVB[267].IN_MaskEn,
	IO 					:= IO_AVB[267],
	HMI 				:= HMI_AVB[267]
	);

	//AVB268 CIP/COP To DRAIN v1.4
	AVB[268](
	IN_ConfigPresent 	:= AVB[268].IN_ConfigPresent,
	IN_Enable 			:= AVB[268].IN_Enable,
	IN_AutoCnd 			:= AVB[268].IN_AutoCnd,
	IN_EnableCnd 		:= AVB[268].IN_EnableCnd,
	IN_Cnd 				:= AVB[268].IN_Cnd,
	IN_FlipEnable 		:= FALSE,
	IN_FlipRequest		:= FALSE,
	IN_FlipTime 		:= T#500ms,
	IN_Reset 			:= VAR_RNS_PBResetEp,
	IN_HMIAutoForce 	:= NOT HMI_SS2P[SS2P_HMI_DeviceEnable].ON,
	IN_ManEn 			:= AVB[268].IN_ManEn,
	IN_MaskEn 			:= AVB[268].IN_MaskEn,
	IO 					:= IO_AVB[268],
	HMI 				:= HMI_AVB[268]
	);

	//AVB273 AIR RINSING VALVE	V4.A.A.1.7.0
	AVB[273](
	IN_ConfigPresent 	:= AVB[273].IN_ConfigPresent,
	IN_Enable 			:= AVB[273].IN_Enable,
	IN_AutoCnd 			:= AVB[273].IN_AutoCnd,
	IN_EnableCnd 		:= AVB[273].IN_EnableCnd,
	IN_Cnd 				:= AVB[273].IN_Cnd,
	IN_FlipEnable 		:= FALSE,
	IN_FlipRequest		:= FALSE,
	IN_FlipTime 		:= T#500ms,
	IN_Reset 			:= VAR_RNS_PBResetEp,
	IN_HMIAutoForce 	:= NOT HMI_SS2P[SS2P_HMI_DeviceEnable].ON,
	IN_ManEn 			:= AVB[273].IN_ManEn,
	IN_MaskEn 			:= AVB[273].IN_MaskEn,
	IO 					:= IO_AVB[273],
	HMI 				:= HMI_AVB[273]
	);

	//AVB294 vrma
	AVB[294](
	IN_ConfigPresent 	:= AVB[294].IN_ConfigPresent,
	IN_Enable 			:= AVB[294].IN_Enable,
	IN_AutoCnd 			:= AVB[294].IN_AutoCnd,
	IN_EnableCnd 		:= AVB[294].IN_EnableCnd,
	IN_Cnd 				:= AVB[294].IN_Cnd,
	IN_FlipEnable 		:= FALSE,
	IN_FlipRequest		:= FALSE,
	IN_FlipTime 		:= T#500ms,
	IN_Reset 			:= VAR_RNS_PBResetEp,
	IN_HMIAutoForce 	:= NOT HMI_SS2P[SS2P_HMI_DeviceEnable].ON,
	IN_ManEn 			:= AVB[294].IN_ManEn,
	IN_MaskEn 			:= AVB[294].IN_MaskEn,
	IO 					:= IO_AVB[294],
	HMI 				:= HMI_AVB[294]
	);

	//VALVES STATUS CONTROL
	VAR_RNS_InletOpen				:= (AVB[261].IN_ConfigPresent AND AVB[261].OUT_OpenedFiltered) AND (AVB[261].OUT_OpenedFiltered OR NOT AVB[261].IN_ConfigPresent);

	VAR_RNS_InletProductIncoming 	:= (AVB[264].OUT_OpenedFiltered OR NOT AVB[264].IN_ConfigPresent) AND VAR_RNS_InletOpen;

	//VALVE FAULT
	VAR_RNS_AVB_ValveFault	:= FALSE;

	FOR VAR_RNS_ForIndex:= MIN_CFG_AVx TO MAX_CFG_AVx DO
		IF AVB[VAR_RNS_ForIndex].IN_ConfigPresent AND AVB[VAR_RNS_ForIndex].OUT_Alarm THEN
			VAR_RNS_AVB_ValveFault	:= TRUE;
		END_IF
	END_FOR

	//INLET CLOSE DUE TO A FAULT
	TMR_TON_InletSafetyDelay.IN := ALR[1512].Active;
	TMR_TON_InletSafetyDelay.PT := T#2s;
	TMR_TON_InletSafetyDelay();

	VAR_RNS_ProductInletSafety		:= TMR_TON_InletSafetyDelay.IN;
	VAR_RNS_ProductInletSafetyDelay	:= TMR_TON_InletSafetyDelay.Q AND AVB[223].OUT_ClosedFiltered;

	//Batteria 203PUB
	IO_203PUB_1.0 := IO_AVB[228].DO_Opened; //DO-02
	IO_203PUB_1.1 := IO_AVB[224].DO_Opened; //DO-01
	IO_203PUB_1.2 := IO_AVB[261].DO_Opened;	//DO-04
	IO_203PUB_1.3 := IO_AVB[234].DO_Opened; //DO-03
	IO_203PUB_1.4 := IO_AVB[268].DO_Opened;	//DO-06
	IO_203PUB_1.5 := IO_AVB[267].DO_Opened;	//DO-05
	IO_203PUB_1.6 := IO_AVB[264].DO_Opened;	//DO-08
	IO_203PUB_1.7 := IO_AVB[294].DO_Opened;	//DO-07

	IO_203PUB_2.0 := FALSE;					//DO-10
	IO_203PUB_2.1 := FALSE;					//DO-09
	IO_203PUB_2.2 := FALSE;					//DO-12
	IO_203PUB_2.3 := FALSE;					//DO-11
	IO_203PUB_2.4 := FALSE;					//DO-14
	IO_203PUB_2.5 := FALSE;					//DO-13
	IO_203PUB_2.6 := FALSE;					//DO-16
	IO_203PUB_2.7 := FALSE;					//DO-15

END_ACTION
```

#### RNS_ModulatingValvesPID.st
```iecst
ACTION RNS_ModulatingValvesPID:
END_ACTION
```

#### RNS_PumpsLogic.st
```iecst
ACTION RNS_PumpsLogic:
	VAR_RNS_PumpEnable 					:= OPS.DataOut.EmergencyOk;
	VAR_RNS_SEQ.Device.PPB209.IN_FixOut	:= (VAR_RNS_FMDProduction OR VAR_RNS_FMDControl) AND PPB[209].IN_ConfigPresent;//vrma
										   //(VAR_RNS_FMDProduction OR VAR_RNS_FMDCip OR VAR_RNS_FMDControl) AND PPB[209].IN_ConfigPresent;//vrma

//	VAR_SetReset(
//	SET1 	:= LSB[210].OUT_OnDelayed AND LSB[299].OUT_OnDelayed,
//	RESET 	:= NOT LSB[210].OUT_OnDelayed);

	VAR_SetReset(
	SET1 	:= LTB[202].OUT_ActValue > 10.0,
	RESET 	:= LTB[202].OUT_ActValue < 5.0);

//PPB209 RINSER RECOVERY PUMP
	PPB[209].IN_Enable 			:= VAR_RNS_PumpEnable;
	PPB[209].IN_AutoCnd 		:= PPB[209].IN_Enable AND VAR_RNS_SEQ.Device.PPB209.IN_FixOut AND VAR_SetReset.Q1;
	PPB[209].IN_AutoSpeed 		:= VAR_RNS_SEQ.Device.PPB209.IN_FixOutValue;
	//	PPB[209].IN_CoastingCmd		:= NOT OPS.DataOut.EnablePump;
END_ACTION
```

#### RNS_PumpsPID.st
```iecst
ACTION RNS_PumpsPID:
	//PPB209 RINSER RECOVERY PUMP MANAGEMENT IN PROD

	IF VAR_RNS_TankLevelTooLow THEN
		VAR_RNS_SEQ.Device.PPB209.IN_FixOutValue := 0.0;
	ELSE
		IF NOT VAR_RNS_TankLevelMedium AND NOT VAR_RNS_TankLevelHigh THEN
			VAR_RNS_SEQ.Device.PPB209.IN_FixOutValue	:= HMI_PAM_1._116;
		ELSIF VAR_RNS_TankLevelMedium AND NOT VAR_RNS_TankLevelHigh THEN
			VAR_RNS_SEQ.Device.PPB209.IN_FixOutValue	:= HMI_PAM_1._117;
		ELSIF VAR_RNS_TankLevelMedium AND VAR_RNS_TankLevelHigh THEN
			VAR_RNS_SEQ.Device.PPB209.IN_FixOutValue	:= HMI_PAM_1._118;
		END_IF
	END_IF

	//Configurazione set point per funzionamento pompa
	HMI_CFG_PAM_1._116 := PPB[209].IN_ConfigPresent;
	HMI_CFG_PAM_1._117 := PPB[209].IN_ConfigPresent;
	HMI_CFG_PAM_1._118 := PPB[209].IN_ConfigPresent;

//	FB_PID_PPB209.IN_ConfigPresent	:= TNK.DataOut.ProdMode AND PTB[290].IN_ConfigPresent;
//	FB_PID_PPB209(
//		IN_ConfigPresent 	:= FB_PID_PPB209.IN_ConfigPresent,
//		IN_ConfigEngValue 	:= TRUE,
//		IN_Reverse 			:= FALSE,
//		IN_Gain 			:= HMI_PAM_D1._085,
//		IN_TI 				:= HMI_PAM_D1._086,
//		IN_TD 				:= HMI_PAM_D1._087,
//		IN_PV 				:= PPB[209].OUT_ActualSpeed,
////		IN_Auto 			:= 0.0,
////		IN_FixOut 			:= ,
//		IN_FixOutValue 		:= HMI_PAM_1._118,
////		IN_IntHold 			:= ,
//		IN_AutoSP 			:= PTB[290].IN_ActualSP,
////		IN_Disv 			:= ,
//		IN_MaxScale 		:= PTB[290].IN_ScaleHIGH,
////		IN_Slew 			:= ,
////		IN_SPSlew 			:= ,
////		IN_MinDev 			:= ,
////		IN_MaxDev 			:= ,
//		IN_OutMin 			:= PPB[209].IN_FrequencyMin,
//		IN_OutMax 			:= PPB[209].IN_FrequencyMax,
//		IN_CycleTime 		:= t#200ms,
//		IN_TIInit 			:= FALSE,
//		IN_TIInitValue 		:= 0.0,
//		HMI 				:= HMI_PID_PPB[209]
//	);

END_ACTION
```

#### RNS_PumpsFB.st
```iecst
ACTION RNS_PumpsFB:
//PPB209 RINSER RECOVERY PUMP
	PPB[209](
	IN_Simulation 		:= FALSE,
	IN_ConfigPresent 	:= PPB[209].IN_ConfigPresent,
	IN_Enable 			:= PPB[209].IN_Enable,
	IN_AutoCnd 			:= PPB[209].IN_AutoCnd,
	IN_AutoSpeed 		:= PPB[209].IN_AutoSpeed,
	IN_Reverse 			:= FALSE,
	IN_FrequencyMin 	:= HMI_PAM_B1._040,
	IN_FrequencyMax 	:= HMI_PAM_B1._041,
	IN_ManEn 			:= TRUE,
	IN_MaskEn 			:= TRUE,
	IN_Reset 			:= VAR_RNS_PBResetEp,
	IN_HMIAutoForce 	:= NOT HMI_SS2P[SS2P_HMI_DeviceEnable].ON,
	IN_QuickStopCmd		:= NOT IO_PPB[209].DI_SafetyEnable,
	IN_JOGMode 			:= FALSE,
	IN_JOGCnd 			:= FALSE,
	IN_CoastingCmd 		:= PPB[209].IN_CoastingCmd,
	IN_FBKDelay 		:= T#1000MS,
	IN_SafetyCtrlEn 	:= FALSE,
	IN_ScaleMax 		:= 100.0,
	HMI_Danfoss 		:= HMI_VFD_PPB[209],
	HMI_Motor 			:= HMI_PPB[209],
	IO_DanfossFC280 			:= IO_VFD_PPB[209],
	IO_MotorFC280 			:= IO_PPB[209]
	);

	HMI_CFG_PAM_B1._040 := PPB[209].IN_ConfigPresent;
	HMI_CFG_PAM_B1._041 := PPB[209].IN_ConfigPresent;
END_ACTION
```

#### RNS_HMI.st
```iecst
ACTION RNS_HMI:
	VAR_RNS_MemPBStart			:= FALSE;
	VAR_RNS_MemPBStop			:= FALSE;
	VAR_RNS_MemPBAbort			:= FALSE;
	VAR_RNS_MemPBSkipForward	:= FALSE;

	//MODE MAN/AUTO
	HMI_RNS_SS2P[SS2P_SelAutoMan].Enable			:= HMI_SS2P[SS2P_HMI_SelEnable].ON AND VAR_RNS_ModeWait;
	HMI_RNS_SS2P[SS2P_SelAutoMan].LampON			:= HMI_RNS_SS2P[SS2P_SelAutoMan].ON;

	//SS2P Production
	HMI_RNS_SS2P[SS2P_SelProduction].Enable			:= HMI_SS2P[SS2P_HMI_SelEnable].ON AND HMI_RNS_SS2P[SS2P_SelAutoMan].ON AND VAR_RNS_ModeWait AND NOT TNK.DataOut.CipMode;
	HMI_RNS_SS2P[SS2P_SelProduction].LampON			:= HMI_RNS_SS2P[SS2P_SelProduction].ON;

	//SS2P Drain
	HMI_RNS_SS2P[SS2P_SelDrain].Enable				:= HMI_SS2P[SS2P_HMI_SelEnable].ON AND HMI_RNS_SS2P[SS2P_SelAutoMan].ON AND VAR_RNS_ModeWait AND NOT TNK.DataOut.CipMode;
	HMI_RNS_SS2P[SS2P_SelDrain].LampON				:= HMI_RNS_SS2P[SS2P_SelDrain].ON;

	//SS2P Cleaning
	HMI_RNS_SS2P[SS2P_SelCIP].Enable				:= HMI_SS2P[SS2P_HMI_SelEnable].ON AND HMI_RNS_SS2P[SS2P_SelAutoMan].ON AND VAR_RNS_ModeWait AND TNK.DataOut.Wait;
	HMI_RNS_SS2P[SS2P_SelCIP].LampON				:= HMI_RNS_SS2P[SS2P_SelCIP].ON;

	//SS2P Control Insercion
	HMI_RNS_SS2P[SS2P_RNS_InsControl].Enable		:= HMI_SS2P[SS2P_HMI_SelEnable].ON AND HMI_RNS_SS2P[SS2P_SelAutoMan].ON AND VAR_RNS_ModeWait AND NOT TNK.DataOut.CipMode;
	HMI_RNS_SS2P[SS2P_RNS_InsControl].LampON		:= HMI_RNS_SS2P[SS2P_RNS_InsControl].ON;

	//SS2P Control Continous
	HMI_RNS_SS2P[SS2P_RNS_ContControl].Enable		:= HMI_SS2P[SS2P_HMI_SelEnable].ON AND HMI_RNS_SS2P[SS2P_SelAutoMan].ON AND VAR_RNS_ModeWait AND NOT TNK.DataOut.CipMode;
	HMI_RNS_SS2P[SS2P_RNS_ContControl].LampON		:= HMI_RNS_SS2P[SS2P_RNS_ContControl].ON;

	//SS2P Bypass Request Manual V4.A.A.1.7.0
	HMI_RNS_SS2P[SS2P_RNS_Bypass].Visibility		:= FALSE;//vrma
	HMI_RNS_SS2P[SS2P_RNS_Bypass].Enable			:= HMI_SS2P[SS2P_HMI_SelEnable].ON AND HMI_RNS_SS2P[SS2P_SelAutoMan].ON AND VAR_RNS_ModeWait AND NOT TNK.DataOut.CipMode;
	HMI_RNS_SS2P[SS2P_RNS_Bypass].LampON			:= HMI_RNS_SS2P[SS2P_RNS_Bypass].ON;

	//PB Mode Start
	VAR_RNS_PBSelectionEnable := HMI_RNS_SS2P[SS2P_SelAutoMan].ON AND
	(HMI_RNS_SS2P[SS2P_SelProduction].ON OR
	((HMI_RNS_SS2P[SS2P_SelDrain].ON OR HMI_RNS_SS2P[SS2P_SelCIP].ON) AND OPS.DataOut.InletGateClosed) OR HMI_RNS_SS2P[SS2P_RNS_ContControl].ON OR HMI_RNS_SS2P[SS2P_RNS_InsControl].ON);

	HMI_RNS_PB[PB_CmdStart].Enable					:= VAR_RNS_PBSelectionEnable AND VAR_RNS_ModeWait;
	HMI_RNS_PB[PB_CmdStart].LampON					:= HMI_RNS_PB[PB_CmdStart].ON;

	//PB Mode Stop
	HMI_RNS_PB[PB_CmdStop].Enable					:= VAR_RNS_PBSelectionEnable AND NOT VAR_RNS_ModeWait;
	HMI_RNS_PB[PB_CmdStop].LampON					:= HMI_RNS_PB[PB_CmdStop].ON;

	//STATUS BAR
	HMI_RNS_State.Sequencer.TextBar[0].Visibility	:= TRUE;
	HMI_RNS_State.Sequencer.TextBar[0].IndexNr		:= FB_RNS_SEQ.IN_Step;
	HMI_RNS_State.Sequencer.TextBar[0].IndexText	:= FB_RNS_SEQ.OUT_HMI_ID;

	HMI_RNS_State.Sequencer.TextBar[1].Visibility	:= FALSE;
	HMI_RNS_State.Sequencer.TextBar[1].IndexNr		:= 0;
	HMI_RNS_State.Sequencer.TextBar[1].IndexText	:= 0;

	//INFO BOX:STEPS
	HMI_RNS_State.Sequencer.InfoBox[0].Visibility			:= FB_RNS_SEQ.OUT_StepTimePr_T>0 OR FB_RNS_SEQ.OUT_StepTimePr_TON>0;
	HMI_RNS_State.Sequencer.InfoBox[0].IndexText			:= '@Lbl_Step@ time';
	HMI_RNS_State.Sequencer.InfoBox[0].Unit					:= 0;
	HMI_RNS_State.Sequencer.InfoBox[0].ProgressVisibility	:= TRUE;
	HMI_RNS_State.Sequencer.InfoBox[0].Progress				:= UINT_TO_REAL(FB_RNS_SEQ.OUT_StepProgressiveTime);
	HMI_RNS_State.Sequencer.InfoBox[0].Preset				:= UINT_TO_REAL(FB_RNS_SEQ.OUT_StepTimePr_TON);
	HMI_RNS_State.Sequencer.InfoBox[0].Actual				:= UINT_TO_REAL(FB_RNS_SEQ.OUT_StepTimeCV_TON);

	HMI_202DSB;

	ComboBoxString(
	IN_ElementsStructure	:= HMI_RNS_Treatments,
	OUT_ComboString			:= ADR(HMI_RNS_TypeCFG)
	);

	(*RNS Multichoice vrma*)
	IF CFG_Par.Rinser.PressureNozzleControlInsertion OR CFG_Par.Rinser.PressureNozzleControlContinous THEN
		HMI_RNS_MultiChoiceMng := 1;
	ELSE
		HMI_RNS_MultiChoiceMng := 0;
	END_IF

	HMI_RNS_PB[PB_RNS_PageUp].Enable	:= VAR_RNS_ActPageData > 0;
	HMI_RNS_PB[PB_RNS_PageUp].LampON := HMI_RNS_PB[PB_RNS_PageUp].ON;

	IF EDGEPOS(HMI_RNS_PB[PB_RNS_PageUp].LampON) THEN
		VAR_RNS_ActPageData := VAR_RNS_ActPageData - 1;
	END_IF

	HMI_RNS_PB[PB_RNS_PageDown].Enable	:= VAR_RNS_ActPageData < VAR_RNS_MaxPageData;
	HMI_RNS_PB[PB_RNS_PageDown].LampON := HMI_RNS_PB[PB_RNS_PageDown].ON;

	IF EDGEPOS(HMI_RNS_PB[PB_RNS_PageDown].LampON) THEN
		VAR_RNS_ActPageData := VAR_RNS_ActPageData + 1;
	END_IF

	IF VAR_RNS_NozzleInLastPage > 0 THEN
		IF VAR_RNS_ActPageData =  VAR_RNS_MaxPageData THEN
			FOR VAR_RNS_IndexVis := 0 TO 14 DO
				VAR_RNS_RnsNozzleData[VAR_RNS_IndexVis + 1 + (VAR_RNS_MaxPageData *15)].Visibility := 	VAR_RNS_IndexVis < VAR_RNS_NozzleInLastPage;
			END_FOR
		ELSE
			VAR_RNS_IndexVis := 0;
		END_IF
	END_IF

	memcpy(ADR(HMI_RNS_NozzleData[1]),ADR(VAR_RNS_RnsNozzleData[1 + (VAR_RNS_ActPageData * 15)]),SIZEOF(HMI_RNS_NozzleData[1]));
	memcpy(ADR(HMI_RNS_NozzleData[2]),ADR(VAR_RNS_RnsNozzleData[2 + (VAR_RNS_ActPageData * 15)]),SIZEOF(HMI_RNS_NozzleData[2]));
	memcpy(ADR(HMI_RNS_NozzleData[3]),ADR(VAR_RNS_RnsNozzleData[3 + (VAR_RNS_ActPageData * 15)]),SIZEOF(HMI_RNS_NozzleData[3]));
	memcpy(ADR(HMI_RNS_NozzleData[4]),ADR(VAR_RNS_RnsNozzleData[4 + (VAR_RNS_ActPageData * 15)]),SIZEOF(HMI_RNS_NozzleData[4]));
	memcpy(ADR(HMI_RNS_NozzleData[5]),ADR(VAR_RNS_RnsNozzleData[5 + (VAR_RNS_ActPageData * 15)]),SIZEOF(HMI_RNS_NozzleData[5]));
	memcpy(ADR(HMI_RNS_NozzleData[6]),ADR(VAR_RNS_RnsNozzleData[6 + (VAR_RNS_ActPageData * 15)]),SIZEOF(HMI_RNS_NozzleData[6]));
	memcpy(ADR(HMI_RNS_NozzleData[7]),ADR(VAR_RNS_RnsNozzleData[7 + (VAR_RNS_ActPageData * 15)]),SIZEOF(HMI_RNS_NozzleData[7]));
	memcpy(ADR(HMI_RNS_NozzleData[8]),ADR(VAR_RNS_RnsNozzleData[8 + (VAR_RNS_ActPageData * 15)]),SIZEOF(HMI_RNS_NozzleData[8]));
	memcpy(ADR(HMI_RNS_NozzleData[9]),ADR(VAR_RNS_RnsNozzleData[9 + (VAR_RNS_ActPageData * 15)]),SIZEOF(HMI_RNS_NozzleData[9]));
	memcpy(ADR(HMI_RNS_NozzleData[10]),ADR(VAR_RNS_RnsNozzleData[10 + (VAR_RNS_ActPageData * 15)]),SIZEOF(HMI_RNS_NozzleData[10]));
	memcpy(ADR(HMI_RNS_NozzleData[11]),ADR(VAR_RNS_RnsNozzleData[11 + (VAR_RNS_ActPageData * 15)]),SIZEOF(HMI_RNS_NozzleData[11]));
	memcpy(ADR(HMI_RNS_NozzleData[12]),ADR(VAR_RNS_RnsNozzleData[12 + (VAR_RNS_ActPageData * 15)]),SIZEOF(HMI_RNS_NozzleData[12]));
	memcpy(ADR(HMI_RNS_NozzleData[13]),ADR(VAR_RNS_RnsNozzleData[13 + (VAR_RNS_ActPageData * 15)]),SIZEOF(HMI_RNS_NozzleData[13]));
	memcpy(ADR(HMI_RNS_NozzleData[14]),ADR(VAR_RNS_RnsNozzleData[14 + (VAR_RNS_ActPageData * 15)]),SIZEOF(HMI_RNS_NozzleData[14]));
	memcpy(ADR(HMI_RNS_NozzleData[15]),ADR(VAR_RNS_RnsNozzleData[15 + (VAR_RNS_ActPageData * 15)]),SIZEOF(HMI_RNS_NozzleData[15]));

	(*RNS Nozzles Data Reset V4.A.A.1.7.0*)
	HMI_RNS_PB[PB_RNS_CounterReset].Visibility := TRUE;
	HMI_RNS_PB[PB_RNS_CounterReset].Enable	:= NOT RNS.DataOut.ContinousControlActive AND NOT RNS.DataOut.InsrtcionControlActive;
	HMI_RNS_PB[PB_RNS_CounterReset].LampON := HMI_RNS_PB[PB_RNS_CounterReset].ON;

	IF HMI_RNS_PB[PB_RNS_CounterReset].LampON THEN
		FOR VAR_RNS_IndexReset := 1 TO 200 DO
			memset(ADR(VAR_RNS_RnsNozzleData[VAR_RNS_IndexReset].ContinousAir),0,SIZEOF(VAR_RNS_RnsNozzleData[VAR_RNS_IndexReset].ContinousAir));
			memset(ADR(VAR_RNS_RnsNozzleData[VAR_RNS_IndexReset].ContinousWater),0,SIZEOF(VAR_RNS_RnsNozzleData[VAR_RNS_IndexReset].ContinousWater));
			memset(ADR(VAR_RNS_RnsNozzleData[VAR_RNS_IndexReset].InsercionAir),0,SIZEOF(VAR_RNS_RnsNozzleData[VAR_RNS_IndexReset].InsercionAir));
			memset(ADR(VAR_RNS_RnsNozzleData[VAR_RNS_IndexReset].InsercionWater),0,SIZEOF(VAR_RNS_RnsNozzleData[VAR_RNS_IndexReset].InsercionWater));
		END_FOR
		VAR_RNS_ContinousAirAlarm	 	:= 0;
		VAR_RNS_ContinousWaterAlarm 	:= 0;
		VAR_RNS_InsercionAirAlarm 		:= 0;
		VAR_RNS_InsercionWaterAlarm		:= 0;
	ELSE
		VAR_RNS_IndexReset := 1;
	END_IF
	(*RNS Nozzles Alarm Detection after control V4.A.A.1.7.0*)
	IF VAR_RNS_SeqActualStep = 81 THEN
		FOR VAR_RNS_IndexAlarm := 1 TO 200 DO
			VAR_RNS_ContinousAirAlarm	 	:= VAR_RNS_ContinousAirAlarm + BOOL_TO_INT(VAR_RNS_RnsNozzleData[VAR_RNS_IndexAlarm].ContinousAir.Alarm);
			VAR_RNS_ContinousWaterAlarm 	:= VAR_RNS_ContinousWaterAlarm + BOOL_TO_INT(VAR_RNS_RnsNozzleData[VAR_RNS_IndexAlarm].ContinousWater.Alarm);
			VAR_RNS_InsercionAirAlarm 		:= VAR_RNS_InsercionAirAlarm + BOOL_TO_INT(VAR_RNS_RnsNozzleData[VAR_RNS_IndexAlarm].InsercionAir.Alarm);
			VAR_RNS_InsercionWaterAlarm		:= VAR_RNS_InsercionWaterAlarm + BOOL_TO_INT(VAR_RNS_RnsNozzleData[VAR_RNS_IndexAlarm].InsercionAir.Alarm);
		END_FOR
	ELSE
		VAR_RNS_IndexAlarm := 1;
	END_IF
	//Added For HMI Recipe problem REMOVE ONCE SOLVED
//	HMI_PAR_1._164 := 480.0;
//	HMI_PAR_1._165 := 400.0;
//	HMI_PAR_1._166 := 350.0;
//	HMI_PAR_1._167 := 260.0;
//	HMI_PAR_1._168 := 5.0;
//	HMI_PAR_1._169 := 30.0;

END_ACTION
```

#### RNS_Alarm.st
```iecst
ACTION RNS_Alarm:
//	ALR[1501].Active	:= VAR_RNS_ModeProduction AND LTB[202].OUT_LowLimit;//vrma CONTROLLA

	ALR[1502].Active	:= LSB[210].OUT_OffDelayed AND VAR_RNS_ModeCip;

	ALR[1506].Active	:= FTB[220].OUT_Alarm OR FTB[270].OUT_Alarm;

	ALR[1513].Active	:= TNK.DataOut.ProdMode AND FSB[201].OUT_Alarm;

	ALR[1512].ActionEn 	:= VAR_RNS_ModeControl OR VAR_RNS_ModeProduction OR VAR_RNS_ModeCop;
	ALR[1512].Active 	:= VAR_RNS_AVB_ValveFault;
	ALR[1514].Active	:= GNS.DataOut.RnsCtrlPistonAlarm;

	ALR[1517].Active	:= _202DSB.OUT_Alarm;

	ALR[1521].ActionEn 	:= VAR_RNS_ModeControl OR VAR_RNS_ModeProduction OR VAR_RNS_ModeCop;
	ALR[1521].Active 	:= AVB[273].OUT_Alarm;

	ALR[1522].ActionEn 	:= VAR_RNS_ModeControl OR VAR_RNS_ModeProduction OR VAR_RNS_ModeCop;
	ALR[1522].Active 	:= AVB[261].OUT_Alarm;

	ALR[1523].Active	:= PPB[209].OUT_OverloadFault;

	ALR[1525].Active	:= PPB[209].OUT_IsolatedFault;

	ALR[1551].Active	:= GNS.DataOut.RnsCtrlDevInserted;

//	ALR[1571].Active	:= VAR_RNS_ModeProduction AND PTB[290].OUT_LowLimit;//vrma CONTROLLA

	ALR[1577].Active	:= VAR_RNS_StepControl; //VAR_RNS_SEQ.Mem.ControlContinous OR VAR_RNS_SEQ.Mem.ControlInsercion;//V4.A.A.1.7.0

	ALR[1578].Active	:= HMI_RNS_SS2P[SS2P_SelAutoMan].LampON;//V4.A.A.1.7.0

	ALR[1586].Active	:= VAR_RNS_WaterFlowLowWarning;//V4.A.A.1.7.0

	ALR[1593].Active	:= PPB[209].OUT_DriveFault;
	ALR[1594].ActionEn 	:= (VAR_RNS_ModeControl OR VAR_RNS_ModeProduction) AND (CFG_Par.Rinser.ExternalRecoverySkid AND VAR_RNS_WaterTreatment);
	ALR[1594].Active := FALSE;
	ALR[1600].Active	:= VAR_RNS_WaterFlowTooLow;//vrma
	ALR[1601].Active 	:= VAR_RNS_SEQ.Mem.ControlContinous OR VAR_RNS_SEQ.Mem.ControlInsercion;//V4.A.A.1.7.0
	ALR[1607].ActionEn 	:= VAR_RNS_ModeProduction;
	ALR[1607].Active 	:= AVB[264].OUT_Alarm OR PI.OPValveFault.3;
	//V4.A.A.1.7.0 New Alarm
	ALR[1608].ActionEn 	:= TRUE;
	ALR[1608].Active 	:= AVB[265].OUT_Alarm OR PI.OPValveFault.4;
	//V4.A.A.1.7.0 New Alarm
	ALR[1609].ActionEn 	:= VAR_RNS_ModeControl OR VAR_RNS_ModeProduction OR VAR_RNS_ModeCop;
	ALR[1609].Active 	:= AVB[266].OUT_Alarm OR PI.OPValveFault.5;
	//V4.A.A.1.7.0 New Alarms
	ALR[1610].Active 	:= (VAR_RNS_ContinousAirAlarm > 0) OR (VAR_RNS_InsercionAirAlarm > 0);
	ALR[1611].Active 	:= (VAR_RNS_ContinousWaterAlarm > 0) OR (VAR_RNS_InsercionWaterAlarm > 0);
	ALR[1612].Active	:= SFT.DataOut.NoBottleNoSprayPistonFault;//vrma test
	ALR[1613].ActionEn	:= VAR_RNS_ModeCip;//vrma test
	ALR[1613].Active 	:= LTB[202].OUT_HighLimit;//vrma test
	ALR[1614].Active	:= LTB[202].OUT_Alarm;//vrma test
	ALR[1615].Active	:= TNK.DataOut.ProdMode AND VAR_RNS_SEQ.Mem.ContainersStop;//vrma
	ALR[1616].Active	:= VAR_RNS_WaterFlowMissing;//vrma

END_ACTION
```

#### RNS_DataOut.st
```iecst
ACTION RNS_DataOut:
	RNS.DataOut.ByPassRequest 					:= VAR_RNS_BypassCommand;
	RNS.DataOut.InsercionRequest				:= NOT VAR_RNS_BypassCommand;
	RNS.DataOut.ByPassed						:= GNS.DataOut.RnsByPassed AND MNM.DataOut.RinserAxisDisabled;//V4.A.A.1.7.0
	RNS.DataOut.AxisDisableRequest 				:= VAR_RNS_BypassCommand;
	RNS.DataOut.InsrtcionDeviceRequest			:= VAR_RNS_SEQ.Mem.InsercionDevice AND VAR_RNS_ControlInsercionRequest;
	RNS.DataOut.ControlInsercionRequestWater 	:= VAR_RNS_SEQ.Mem.ControlInsercion AND VAR_RNS_SEQ.Mem.WaterTreatmentControl;
	RNS.DataOut.ControlInsercionRequestAir	 	:= VAR_RNS_SEQ.Mem.ControlInsercion AND VAR_RNS_SEQ.Mem.AirTreatmentControl;
	RNS.DataOut.ControlContinousRequestWater	:= VAR_RNS_SEQ.Mem.ControlContinous AND VAR_RNS_SEQ.Mem.WaterTreatmentControl;
	RNS.DataOut.ControlContinousRequestAir		:= VAR_RNS_SEQ.Mem.ControlContinous AND VAR_RNS_SEQ.Mem.AirTreatmentControl;
	RNS.DataOut.InsrtcionControlActive 			:= VAR_RNS_FMDControl AND GNS.DataOut.RnsCtrlDevInserted AND MNM.DataOut.RnsSpeedReqReached AND SFT.DataOut.MachineEmpty;
	RNS.DataOut.ContinousControlActive			:= VAR_RNS_FMDControl AND MNM.DataOut.RnsSpeedReqReached AND SFT.DataOut.MachineEmpty;
	RNS.DataOut.ProdMode 						:= VAR_RNS_SEQ.ITC.WTT_ProductionRunning;
	RNS.DataOut.ProductRequest 					:= VAR_RNS_SEQ.ITC.WTT_ProductRequest OR AVB[228].IN_AutoCnd OR AVB[266].IN_AutoCnd;//V4.A.A.1.7.0
	RNS.DataOut.CopMode							:= VAR_RNS_SEQ.Mem.CopAfterCipRequest;//V4.A.A.1.7.0
	RNS.DataOut.StepCounterRequest				:= RNS.DataOut.ContinousControlActive OR RNS.DataOut.InsrtcionControlActive OR VAR_RNS_SeqPermanent.SeqActualStep = 14;
	RNS.DataOut.FixSpeedRequest					:= VAR_RNS_SEQ.Mem.SpeedReductionControl OR (HMI_RNS_SS2P[SS2P_SelAutoMan].ON AND HMI_RNS_SS2P[SS2P_RNS_ContControl].ON AND VAR_RNS_MemPBStart);
	RNS.DataOut.MachineStart					:= RNS.DataOut.FixSpeedRequest;
	RNS.DataOut.MachineStop						:= NOT RNS.DataOut.FixSpeedRequest;
	RNS.DataOut.CipMode							:= VAR_RNS_FMDCip;
	RNS.DataOut.NoBottleNoSprayInsercion		:= VAR_RNS_SEQ.Mem.NoBoNoSprayInsercion;//vrma test
	RNS.DataOut.ContainerStop					:= VAR_RNS_SEQ.Mem.ContainersStop;
	RNS.DataOut.CipDrainEnd						:= VAR_RNS_StepCipEnded;

	RNS.DataOut.RunOnlyRinserAxisRequest		:= VAR_RNS_SeqPermanent.SeqMode1.7 AND NOT DOS.DataOut.CipMode;
	RNS.DataOut.RunWithHemaReq		            := VAR_RNS_SeqPermanent.SeqMode1.7 AND DOS.DataOut.CipMode;

	IF VAR_RNS_SEQ.Mem.InsercionDevice OR VAR_RNS_ModeCip THEN
		RNS.DataOut.FixSpeedValue					:= HMI_PAM_1._014;
	ELSE
		RNS.DataOut.FixSpeedValue					:= HMI_PAM_1._015;
	END_IF

END_ACTION
```

#### RNS_Hardware_CFG.st
```iecst
ACTION RNS_Hardware_CFG:
	(*****MACHINE*****)

	(*****DIGITAL*****)
	FSB[201].IN_ConfigPresent 	:= TRUE;
	FSB[201].IN_OnDelay			:= T#5ms;
	FSB[201].IN_OffDelay		:= T#25s;

	FSB[220].IN_ConfigPresent 	:= TRUE;
	FSB[220].IN_OnDelay			:= T#1s;
	FSB[220].IN_OffDelay		:= T#5s;

	(*****VALVES*****)
	AVB[224].IN_ConfigPresent				:= TRUE;
	AVB[224].IN_ConfigType 					:= 0;
	AVB[224].IN_Simulation 					:= FALSE;
	AVB[224].IN_ConfigPositionSensorOpened 	:= TRUE;
	AVB[224].IN_ConfigPositionSensorClosed 	:= TRUE;
	AVB[224].IN_StrokeTime 					:= T#5s;

	AVB[228].IN_ConfigPresent				:= TRUE;
	AVB[228].IN_ConfigType 					:= 0;
	AVB[228].IN_Simulation 					:= FALSE;
	AVB[228].IN_ConfigPositionSensorOpened 	:= TRUE;
	AVB[228].IN_ConfigPositionSensorClosed 	:= TRUE;
	AVB[228].IN_StrokeTime 					:= T#2s;

	AVB[234].IN_ConfigPresent				:= TRUE;
	AVB[234].IN_ConfigType 					:= 0;
	AVB[234].IN_Simulation 					:= FALSE;
	AVB[234].IN_ConfigPositionSensorOpened 	:= TRUE;
	AVB[234].IN_ConfigPositionSensorClosed 	:= TRUE;
	AVB[234].IN_StrokeTime 					:= T#2s;

	AVB[261].IN_ConfigPresent				:= TRUE;
	AVB[261].IN_ConfigType 					:= 0;
	AVB[261].IN_Simulation 					:= FALSE;
	AVB[261].IN_ConfigPositionSensorOpened 	:= TRUE;
	AVB[261].IN_ConfigPositionSensorClosed 	:= TRUE;
	AVB[261].IN_StrokeTime 					:= T#2s;

	AVB[264].IN_ConfigPresent				:= TRUE;
	AVB[264].IN_ConfigType 					:= 0;
	AVB[264].IN_Simulation 					:= FALSE;
	AVB[264].IN_ConfigPositionSensorOpened 	:= TRUE;
	AVB[264].IN_ConfigPositionSensorClosed 	:= TRUE;
	AVB[264].IN_StrokeTime 					:= T#5s;

	AVB[265].IN_ConfigPresent				:= FALSE;
	AVB[265].IN_ConfigType 					:= 0;
	AVB[265].IN_Simulation 					:= FALSE;
	AVB[265].IN_ConfigPositionSensorOpened 	:= TRUE;
	AVB[265].IN_ConfigPositionSensorClosed 	:= TRUE;
	AVB[265].IN_StrokeTime 					:= T#4s;

	AVB[266].IN_ConfigPresent				:= FALSE;
	AVB[266].IN_ConfigType 					:= 0;
	AVB[266].IN_Simulation 					:= FALSE;
	AVB[266].IN_ConfigPositionSensorOpened 	:= TRUE;
	AVB[266].IN_ConfigPositionSensorClosed 	:= TRUE;
	AVB[266].IN_StrokeTime 					:= T#2s;

	AVB[267].IN_ConfigPresent				:= TRUE;
	AVB[267].IN_ConfigType 					:= 0;
	AVB[267].IN_Simulation 					:= FALSE;
	AVB[267].IN_ConfigPositionSensorOpened 	:= TRUE;
	AVB[267].IN_ConfigPositionSensorClosed 	:= TRUE;
	AVB[267].IN_StrokeTime 					:= T#2s;

	AVB[268].IN_ConfigPresent				:= TRUE;
	AVB[268].IN_ConfigType 					:= 0;
	AVB[268].IN_Simulation 					:= FALSE;
	AVB[268].IN_ConfigPositionSensorOpened 	:= TRUE;
	AVB[268].IN_ConfigPositionSensorClosed 	:= TRUE;
	AVB[268].IN_StrokeTime 					:= T#2s;

	AVB[273].IN_ConfigPresent				:= FALSE;
	AVB[273].IN_ConfigType 					:= 0;
	AVB[273].IN_Simulation 					:= FALSE;
	AVB[273].IN_ConfigPositionSensorOpened 	:= FALSE;
	AVB[273].IN_ConfigPositionSensorClosed 	:= FALSE;
	AVB[273].IN_StrokeTime 					:= T#2s;

	AVB[294].IN_ConfigPresent				:= TRUE;//vrma
	AVB[294].IN_ConfigType 					:= 0;
	AVB[294].IN_Simulation 					:= FALSE;
	AVB[294].IN_ConfigPositionSensorOpened 	:= TRUE;
	AVB[294].IN_ConfigPositionSensorClosed 	:= TRUE;
	AVB[294].IN_StrokeTime 					:= T#2s;

	(*****PUMPS*****)
	PPB[209].IN_ConfigPresent	:= TRUE;
	PPB[209].IN_Reverse			:= FALSE;

	(*****ANALOG*****)
	FTB[201].IN_ConfigPresent 	:= FALSE;
	FTB[201].IN_Simulation 		:= FALSE;
	FTB[201].IN_0_20mA 			:= TRUE;
	FTB[201].IN_ConfigPopup		:= TRUE;
	FTB[201].IN_FaultOutMode 	:= 0;
	FTB[201].IN_EngScale 		:= FALSE;
	FTB[201].IN_ScaleLOW		:= 0.0;
	FTB[201].IN_ScaleHIGH		:= 800.0;

	FTB[202].IN_ConfigPresent 	:= TRUE;
	FTB[202].IN_Simulation 		:= FALSE;
	FTB[202].IN_0_20mA 			:= TRUE;
	FTB[202].IN_ConfigPopup		:= TRUE;
	FTB[202].IN_FaultOutMode 	:= 0;
	FTB[202].IN_EngScale 		:= FALSE;
	FTB[202].IN_ScaleLOW		:= 0.0;
	FTB[202].IN_ScaleHIGH		:= 400.0;

	PTB[220].IN_ConfigPresent 	:= TRUE;
	PTB[220].IN_Simulation 		:= FALSE;
	PTB[220].IN_0_20mA 			:= TRUE;
	PTB[220].IN_ConfigPopup		:= TRUE;
	PTB[220].IN_FaultOutMode 	:= 0;
	PTB[220].IN_EngScale 		:= FALSE;
	PTB[220].IN_ScaleLOW		:= -1.0;
	PTB[220].IN_ScaleHIGH		:= 10.0;

	PTB[270].IN_ConfigPresent 	:= FALSE;
	PTB[270].IN_Simulation 		:= FALSE;
	PTB[270].IN_0_20mA 			:= TRUE;
	PTB[270].IN_ConfigPopup		:= TRUE;
	PTB[270].IN_FaultOutMode 	:= 0;
	PTB[270].IN_EngScale 		:= FALSE;
	PTB[270].IN_ScaleLOW		:= -1.0;
	PTB[270].IN_ScaleHIGH		:= 10.0;

	PTB[290].IN_ConfigPresent 	:= TRUE;//vrma
	PTB[290].IN_Simulation 		:= FALSE;
	PTB[290].IN_0_20mA 			:= TRUE;
	PTB[290].IN_ConfigPopup		:= TRUE;
	PTB[290].IN_FaultOutMode 	:= 0;
	PTB[290].IN_EngScale 		:= FALSE;
	PTB[290].IN_ScaleLOW		:= -1.0;
	PTB[290].IN_ScaleHIGH		:= 10.0;

	LTB[202].IN_ConfigPresent 	:= TRUE;//vrma
	LTB[202].IN_Simulation 		:= FALSE;
	LTB[202].IN_0_20mA 			:= TRUE;
	LTB[202].IN_ConfigPopup		:= TRUE;
	LTB[202].IN_FaultOutMode 	:= 0;
	LTB[202].IN_EngScale 		:= FALSE;
	LTB[202].IN_ScaleLOW		:= 0.0;
	LTB[202].IN_ScaleHIGH		:= 100.0;

END_ACTION
```

### Package Logical/12_MAU - Machine Auxiliary: funzioni macchina ausiliarie

### Program Logical/12_MAU/1280_SafetyCheck/MAU_SafetyCheck (IEC) - MAU_SafetyCheck Main Program - C#7 - 20.8ms

#### Cyclic.st - Cyclic code
```iecst
PROGRAM _CYCLIC
	CMD_SafetyRemoteControl.Password := HMI_SL_Info.Password;

	TMR_TON_Read(
	IN := VAR_SafeRemoteControl_Step = SafeLogic_Wait,
	PT := T#5s
	); //Read SAFE PLC info every 5s

	CASE VAR_SafeRemoteControl_Step OF
		SafeLogic_Wait: //Wait
			IF TMR_TON_Read.Q THEN					//SafeLogic_CMD_ReadStatus;
				VAR_SafeRemoteControl_Step := SafeLogic_ReadOsStatus;
			ELSIF HMI_SL_PB.Ack_SK.ON THEN			//SafeKey acknoledge
				VAR_SafeRemoteControl_Step := SafeLogic_Ack_SK;
			ELSIF HMI_SL_PB.Ack1UdId.ON THEN		//1 UDID acknoledge
				VAR_SafeRemoteControl_Step := SafeLogic_Ack1UdId;
			ELSIF HMI_SL_PB.Ack2UdId.ON THEN		//2 UDID acknoledge
				VAR_SafeRemoteControl_Step := SafeLogic_Ack2UdId;
			ELSIF HMI_SL_PB.Ack3UdId.ON THEN		//3 UDID acknoledge
				VAR_SafeRemoteControl_Step := SafeLogic_Ack3UdId;
			ELSIF HMI_SL_PB.Ack4UdId.ON THEN		//4 UDID acknoledge
				VAR_SafeRemoteControl_Step := SafeLogic_Ack4UdId;
			ELSIF HMI_SL_PB.AckMore4UdId.ON THEN	//4+ UDID acknoledge
				VAR_SafeRemoteControl_Step := SafeLogic_AckMore4UdId;
			ELSIF HMI_SL_PB.AckFW.ON THEN			//Firmware acknoledge
				VAR_SafeRemoteControl_Step := SafeLogic_Ack_FW;
			ELSIF HMI_SL_PB.LedTest.ON THEN			//Test LED
				VAR_SafeRemoteControl_Step := SafeLogic_LedTest;
			ELSIF HMI_SL_PB.Scan.ON THEN			//Scan
				VAR_SafeRemoteControl_Step := SafeLogic_Scan;
			END_IF

		SafeLogic_ReadOsStatus:
			// Init address device to read
			VAR_SafetyDeviceAdress := 'IF3.ST3';

			// Init index and subindex to read : SafeOSState
			VAR_Index		:= 16#2000;
			VAR_Subindex 	:= 16#11;

			// Reading start
			FB_RemoteEplSDORead(
			enable		:= TRUE,
			pDevice		:= ADR(VAR_SafetyDeviceAdress),
			node		:= 3,  //SafeLOGIC EPL Address
			index		:= VAR_Index,
			subindex	:= VAR_Subindex,
			pData		:= ADR(VAR_SafeOSState),
			datalen		:= SIZEOF(VAR_SafeOSState)
			);

			VAR_CPUSafetyNotFound := (FB_RemoteEplSDORead.status = 20925);

			IF FB_RemoteEplSDORead.status <> ERR_FUB_BUSY THEN
				VAR_SafeRemoteControl_Step := SafeLogic_CMD_ReadStatus;
			END_IF

		SafeLogic_CMD_ReadStatus:	//REQUEST SAFE PLC info
			CMD_SafetyRemoteControl.Command	:= 16#200;
			CMD_SafetyRemoteControl.Number	:= 1;
			CMD_SafetyRemoteControl.Data	:= 0;

			FB_RemoteEplSDOWrite(
			enable		:= TRUE,
			pDevice		:= ADR(VAR_SafetyDeviceAdress),
			node		:= 3,
			index		:= 16#2406,
			subindex	:= 16#1,
			pData		:= ADR(CMD_SafetyRemoteControl),
			datalen		:= 22
			);

			IF FB_RemoteEplSDOWrite.status <> ERR_FUB_BUSY THEN
				VAR_SafeRemoteControl_Step := SafeLogic_ReadCRC;
			END_IF

		SafeLogic_ReadCRC: //CRC
			FB_RemoteEplSDORead(
			enable		:= TRUE,
			pDevice		:= ADR(VAR_SafetyDeviceAdress),
			node		:= 3,
			index		:= 16#2000,
			subindex	:= 16#8,
			pData		:= ADR(VAR_SafeCRC),
			datalen		:= SIZEOF(VAR_SafeCRC)
			);

			IF FB_RemoteEplSDORead.status <> ERR_FUB_BUSY THEN
				VAR_SafeRemoteControl_Step := SafeLogic_ReadTime;
			END_IF

		SafeLogic_ReadTime: //Date
			FB_RemoteEplSDORead(
			enable		:= TRUE,
			pDevice		:= ADR(VAR_SafetyDeviceAdress),
			node		:= 3,
			index		:= 16#2000,
			subindex	:= 16#9,
			pData		:= ADR(VAR_SafeTime),
			datalen		:= SIZEOF(VAR_SafeTime)
			);

			IF FB_RemoteEplSDORead.status <> ERR_FUB_BUSY THEN
				VAR_SafeRemoteControl_Step := SafeLogic_ReadAuthor;
			END_IF

		SafeLogic_ReadAuthor: //Author
			FB_RemoteEplSDORead(
			enable		:= TRUE,
			pDevice		:= ADR(VAR_SafetyDeviceAdress),
			node		:= 3,
			index		:= 16#2000,
			subindex	:= 16#D,
			pData		:= ADR(VAR_SafeAuthor),
			datalen		:= SIZEOF(VAR_SafeAuthor)
			);

			IF FB_RemoteEplSDORead.status <> ERR_FUB_BUSY THEN
				VAR_NoUpdateStatus		:= TRUE;
				VAR_SafeRemoteControl_Step	:= SafeLogic_ReadStatus;
			END_IF

		SafeLogic_ReadStatus: //Status
			FB_RemoteEplSDORead(
			enable		:= TRUE,
			pDevice		:= ADR(VAR_SafetyDeviceAdress),
			node		:= 3,
			index		:= 16#2406,
			subindex	:= 16#2,
			pData		:= ADR(VAR_StatusSafetyRemoteControl),
			datalen		:= SIZEOF(VAR_StatusSafetyRemoteControl)
			);

			IF FB_RemoteEplSDORead.status <> ERR_FUB_BUSY THEN
				VAR_StatusSafetyScanning		:= VAR_StatusSafetyRemoteControl.Scanning;
				VAR_StatusSafetySafeKeyChanged	:= VAR_StatusSafetyRemoteControl.SafeKeyChanged;
				VAR_StatusSafetyNbOfUdId		:= VAR_StatusSafetyRemoteControl.NumberOfUdIdMismatches;
				VAR_StatusSafetyNbOfDiffFW		:= VAR_StatusSafetyRemoteControl.NumberOfDiffFirmware;

				IF VAR_NoUpdateStatus THEN
					VAR_NoUpdateStatus						:= FALSE;
					VAR_StatusSafetyRemoteControl.Status	:= 16#FF;
				END_IF

				VAR_SafeRemoteControl_Step	:= SafeLogic_Wait;
			END_IF

		SafeLogic_AckMore4UdId: //Ackowledge more than 4 UDID mismatches
			CMD_SafetyRemoteControl.Command	:= 16#100;
			CMD_SafetyRemoteControl.Number	:= 16#20;
			CMD_SafetyRemoteControl.Data	:= 16#20;

			VAR_SafeRemoteControl_Step		:= SafeLogic_CMD_Write;

		SafeLogic_Ack4UdId: //Ackowledge 4 UDID mismatches
			CMD_SafetyRemoteControl.Command	:= 16#100;
			CMD_SafetyRemoteControl.Number	:= 16#30;
			CMD_SafetyRemoteControl.Data	:= 16#30;

			VAR_SafeRemoteControl_Step		:= SafeLogic_CMD_Write;

		SafeLogic_Ack3UdId: //Ackowledge 3 UDID mismatches
			CMD_SafetyRemoteControl.Command	:= 16#100;
			CMD_SafetyRemoteControl.Number	:= 16#40;
			CMD_SafetyRemoteControl.Data	:= 16#40;

			VAR_SafeRemoteControl_Step		:= SafeLogic_CMD_Write;

		SafeLogic_Ack2UdId: //Ackowledge 2 UDID mismatches
			CMD_SafetyRemoteControl.Command	:= 16#100;
			CMD_SafetyRemoteControl.Number	:= 16#50;
			CMD_SafetyRemoteControl.Data	:= 16#50;

			VAR_SafeRemoteControl_Step		:= SafeLogic_CMD_Write;

		SafeLogic_Ack1UdId: //Ackowledge 1 UDID mismatches
			CMD_SafetyRemoteControl.Command	:= 16#100;
			CMD_SafetyRemoteControl.Number	:= 16#60;
			CMD_SafetyRemoteControl.Data	:= 16#60;

			VAR_SafeRemoteControl_Step		:= SafeLogic_CMD_Write;

		SafeLogic_Ack_FW: //FW-ACKN, acknowledge a new firmware versions
			CMD_SafetyRemoteControl.Command	:= 16#100;
			CMD_SafetyRemoteControl.Number	:= 16#100;
			CMD_SafetyRemoteControl.Data	:= 16#100;

			VAR_SafeRemoteControl_Step		:= SafeLogic_CMD_Write;

		SafeLogic_Ack_SK: //SK-XCHG, acknowledge a SafeKEY exchange
			CMD_SafetyRemoteControl.Command	:= 16#100;
			CMD_SafetyRemoteControl.Number	:= 16#200;
			CMD_SafetyRemoteControl.Data	:= 16#200;

			VAR_SafeRemoteControl_Step		:= SafeLogic_CMD_Write;

		SafeLogic_LedTest: //TEST, start an LED test (5s)
			CMD_SafetyRemoteControl.Command	:= 16#100;
			CMD_SafetyRemoteControl.Number	:= 16#1000;
			CMD_SafetyRemoteControl.Data	:= 16#1000;

			VAR_SafeRemoteControl_Step		:= SafeLogic_CMD_Write;

		SafeLogic_Scan: //SCAN, start a system scan
			CMD_SafetyRemoteControl.Command	:= 16#100;
			CMD_SafetyRemoteControl.Number	:= 16#2000;
			CMD_SafetyRemoteControl.Data	:= 16#2000;

			VAR_SafeRemoteControl_Step		:= SafeLogic_CMD_Write;

		SafeLogic_CMD_Write: //Send command to Safety CPU
			FB_RemoteEplSDOWrite(
			enable		:= TRUE,
			pDevice		:= ADR(VAR_SafetyDeviceAdress),
			node		:= 3,
			index		:= 16#2406,
			subindex	:= 16#1,
			pData		:= ADR(CMD_SafetyRemoteControl),
			datalen		:= 22
			);

			IF FB_RemoteEplSDOWrite.status <> ERR_FUB_BUSY THEN
				HMI_SL_PB.Ack_SK.ON			:= FALSE; //Acknoledge SafeKey
				HMI_SL_PB.Ack1UdId.ON		:= FALSE; //Acknoledge 1 UDID
				HMI_SL_PB.Ack2UdId.ON		:= FALSE; //Acknoledge 2 UDID
				HMI_SL_PB.Ack3UdId.ON		:= FALSE; //Acknoledge 3 UDID
				HMI_SL_PB.Ack4UdId.ON		:= FALSE; //Acknoledge 4 UDID
				HMI_SL_PB.AckMore4UdId.ON	:= FALSE; //Acknoledge 4+ UDID
				HMI_SL_PB.AckFW.ON			:= FALSE; //Acknoledge Firmware
				HMI_SL_PB.LedTest.ON		:= FALSE; //Test LED
				HMI_SL_PB.Scan.ON			:= FALSE; //Scan
				VAR_SafeRemoteControl_Step	:= SafeLogic_ReadStatus;
			END_IF

	END_CASE

	(************************************************************************************************************************)
	(*************************************************  DISPLAY MANAGEMENT  *************************************************)
	(************************************************************************************************************************)
	IF VAR_SafeRemoteControl_Step = SafeLogic_Wait THEN
		//SafeCRC in string
		HMI_SL_Info.CRC := VAR_SafeCRC;

		//SafeTime in string
		DT_TO_DTStructure(VAR_SafeTime, ADR(VAR_SafeTime_DTStruct));
		itoa(VAR_SafeTime_DTStruct.day, ADR(VAR_Temp));
		HMI_SL_Info.Date := VAR_Temp;
		strcat(ADR(HMI_SL_Info.Date), ADR('/'));
		itoa(VAR_SafeTime_DTStruct.month, ADR(VAR_Temp));
		strcat(ADR(HMI_SL_Info.Date), ADR(VAR_Temp));
		strcat(ADR(HMI_SL_Info.Date), ADR('/'));
		itoa(VAR_SafeTime_DTStruct.year, ADR(VAR_Temp));
		VAR_Temp := RIGHT(VAR_Temp,2);
		strcat(ADR(HMI_SL_Info.Date), ADR(VAR_Temp));
		strcat(ADR(HMI_SL_Info.Date), ADR('  '));
		itoa(VAR_SafeTime_DTStruct.hour, ADR(VAR_Temp));
		strcat(ADR(HMI_SL_Info.Date), ADR(VAR_Temp));
		strcat(ADR(HMI_SL_Info.Date), ADR(':'));
		itoa(VAR_SafeTime_DTStruct.minute, ADR(VAR_Temp));
		strcat(ADR(HMI_SL_Info.Date), ADR(VAR_Temp));

		//Safe Author
		HMI_SL_Info.Author				:= VAR_SafeAuthor;

		//Remote Control Status
		HMI_SL_Info.RemoteCtrlStatus	:= VAR_StatusSafetyRemoteControl.Status;

		//Safe Status ID
		HMI_SL_Info.IDMissed := '';
		memset(ADR(VAR_ModuleSafetyMissing), 0, SIZEOF(VAR_ModuleSafetyMissing));
		IF NOT(VAR_SafeOSState = cRUN_SAFE) OR NOT SI_SafeLogicModuleOk THEN
			FOR j := 0 TO ((SIZEOF(VAR_ModuleSafetyMissing) / SIZEOF(VAR_ModuleSafetyMissing[0])) - 1) DO
				VAR_ModuleSafetyMissing[j] := TRUE;
			END_FOR
		END_IF

		IF VAR_StatusSafetyRemoteControl.NumberOfMissingModules <> 0 THEN //Module missing
			FOR i := 0 TO 15 DO
				FOR j := 0 TO 7 DO
					IF BIT_TST(VAR_StatusSafetyRemoteControl.MissingModules[i], j) THEN
						IF strcmp(ADR(HMI_SL_Info.IDMissed), ADR("")) <> 0 THEN
							strcat(ADR(HMI_SL_Info.IDMissed), ADR('/'));
						END_IF
						itoa(VAR_StatusSafetyRemoteControl.SAddr[i * 8 + j], ADR(VAR_Temp));
						VAR_ModuleSafetyMissing[VAR_StatusSafetyRemoteControl.SAddr[i * 8 + j]] := TRUE;
						strcat(ADR(HMI_SL_Info.IDMissed), ADR(VAR_Temp));
					END_IF
				END_FOR
			END_FOR
		END_IF

		HMI_SL_Info.IDMismatches := '';
		IF VAR_StatusSafetyRemoteControl.NumberOfUdIdMismatches <> 0 THEN //Module mismatches
			FOR i := 0 TO 15 DO
				FOR j := 0 TO 7 DO
					IF BIT_TST(VAR_StatusSafetyRemoteControl.UdIdMismatches[i], j) THEN
						IF strcmp(ADR(HMI_SL_Info.IDMismatches), ADR("")) <> 0 THEN
							strcat(ADR(HMI_SL_Info.IDMismatches), ADR('/'));
						END_IF
						itoa(VAR_StatusSafetyRemoteControl.SAddr[i * 8 + j], ADR(VAR_Temp));
						strcat(ADR(HMI_SL_Info.IDMismatches), ADR(VAR_Temp));
					END_IF
				END_FOR
			END_FOR
		END_IF

		HMI_SL_Info.IDDiffFirmware := '';
		IF VAR_StatusSafetyRemoteControl.NumberOfDiffFirmware <> 0 THEN //Module Update
			FOR i := 0 TO 15 DO
				FOR j := 0 TO 7 DO
					IF BIT_TST(VAR_StatusSafetyRemoteControl.DiffFirmware[i], j) THEN
						IF strcmp(ADR(HMI_SL_Info.IDDiffFirmware), ADR("")) <> 0 THEN
							strcat(ADR(HMI_SL_Info.IDDiffFirmware), ADR('/'));
						END_IF
						itoa(VAR_StatusSafetyRemoteControl.SAddr[i * 8 + j], ADR(VAR_Temp));
						strcat(ADR(HMI_SL_Info.IDDiffFirmware), ADR(VAR_Temp));
					END_IF
				END_FOR
			END_FOR
		END_IF

		// Status Text - FAIL LED
		IF (VAR_StatusSafetyRemoteControl.FailSafe <> cFAIL_SAFE_OK) THEN
			HMI_SL_Info.Led.FAIL := 2;
		ELSIF (VAR_StatusSafetyRemoteControl.OpenSafetyState = 0) THEN
			HMI_SL_Info.Led.FAIL := 0;
		ELSIF (VAR_StatusSafetyRemoteControl.OpenSafetyState = 1) THEN
			HMI_SL_Info.Led.FAIL := 1;
		END_IF

		// Status text - FW-ACKN_LED
		IF (VAR_StatusSafetyRemoteControl.SafeKeyChanged = 0 AND VAR_StatusSafetyRemoteControl.NumberOfDiffFirmware = 0) THEN
			HMI_SL_Info.Led.FW_ACKN := 10;
		ELSIF (VAR_StatusSafetyRemoteControl.SafeKeyChanged = 1) THEN
			HMI_SL_Info.Led.FW_ACKN := 1;
		ELSIF (VAR_StatusSafetyRemoteControl.NumberOfDiffFirmware <> 0) THEN
			HMI_SL_Info.Led.FW_ACKN := 2;
		END_IF

		// Status text - MXCHG_LED
		IF (VAR_StatusSafetyRemoteControl.LedTestActive = 1) THEN
			HMI_SL_Info.Led.MXCHG := 40;
		ELSIF (VAR_StatusSafetyRemoteControl.Scanning = 1) THEN
			HMI_SL_Info.Led.MXCHG := 30;
		ELSIF (VAR_StatusSafetyRemoteControl.NumberOfUdIdMismatches = 1) THEN
			HMI_SL_Info.Led.MXCHG := 1;
		ELSIF (VAR_StatusSafetyRemoteControl.NumberOfUdIdMismatches = 2) THEN
			HMI_SL_Info.Led.MXCHG := 2;
		ELSIF (VAR_StatusSafetyRemoteControl.NumberOfUdIdMismatches = 3) THEN
			HMI_SL_Info.Led.MXCHG := 3;
		ELSIF (VAR_StatusSafetyRemoteControl.NumberOfUdIdMismatches = 4) THEN
			HMI_SL_Info.Led.MXCHG := 4;
		ELSIF (VAR_StatusSafetyRemoteControl.NumberOfUdIdMismatches > 4) THEN
			HMI_SL_Info.Led.MXCHG := 5;
		ELSIF (VAR_StatusSafetyRemoteControl.NumberOfMissingModules <> 0) THEN
			HMI_SL_Info.Led.MXCHG := 20;
		ELSIF (VAR_StatusSafetyRemoteControl.NumberOfUdIdMismatches = 0) THEN
			HMI_SL_Info.Led.MXCHG := 10;
		END_IF

		// Status text - RE_LED
		HMI_SL_Info.Led.RE := VAR_StatusSafetyRemoteControl.SafeOSstate;
	END_IF

	VAR_AllowedSafeButton	:= NOT HMI_SL_PB.Ack_SK.LampON			AND NOT HMI_SL_PB.Ack1UdId.LampON	AND NOT HMI_SL_PB.Ack2UdId.LampON		AND
								NOT HMI_SL_PB.Ack3UdId.LampON		AND NOT HMI_SL_PB.Ack4UdId.LampON	AND NOT HMI_SL_PB.AckMore4UdId.LampON	AND
								NOT HMI_SL_PB.AckFW.LampON			AND NOT	HMI_SL_PB.LedTest.LampON	AND NOT HMI_SL_PB.Scan.LampON			AND
								memcmp(ADR(HMI_SL_Info.Password),	ADR(CST_SafePasswordBlank),			SIZEOF(HMI_SL_Info.Password)) <> 0		AND
								memcmp(ADR(HMI_SL_Info.Password),	ADR(CST_SafePasswordNull),			SIZEOF(HMI_SL_Info.Password)) <> 0		AND VAR_StatusSafetyRemoteControl.Status = 255;

	HMI_SL_PB.Ack_SK.Enable			:= (VAR_StatusSafetyScanning = 0	OR (VAR_StatusSafetyScanning = 1		AND HMI_SL_Info.Led.FAIL = 2		AND HMI_SL_Info.Led.RE <> 0))		AND VAR_StatusSafetySafeKeyChanged = 1	AND VAR_AllowedSafeButton;
	HMI_SL_PB.Ack1UdId.Enable		:= VAR_StatusSafetyScanning = 0		AND VAR_StatusSafetySafeKeyChanged = 0	AND VAR_StatusSafetyNbOfUdId = 1	AND VAR_AllowedSafeButton;
	HMI_SL_PB.Ack2UdId.Enable		:= VAR_StatusSafetyScanning = 0		AND VAR_StatusSafetySafeKeyChanged = 0	AND VAR_StatusSafetyNbOfUdId = 2	AND VAR_AllowedSafeButton;
	HMI_SL_PB.Ack3UdId.Enable		:= VAR_StatusSafetyScanning = 0		AND VAR_StatusSafetySafeKeyChanged = 0	AND VAR_StatusSafetyNbOfUdId = 3	AND VAR_AllowedSafeButton;
	HMI_SL_PB.Ack4UdId.Enable		:= VAR_StatusSafetyScanning = 0		AND VAR_StatusSafetySafeKeyChanged = 0	AND VAR_StatusSafetyNbOfUdId = 4	AND VAR_AllowedSafeButton;
	HMI_SL_PB.AckMore4UdId.Enable	:= VAR_StatusSafetyScanning = 0		AND VAR_StatusSafetySafeKeyChanged = 0	AND VAR_StatusSafetyNbOfUdId > 4	AND VAR_AllowedSafeButton;
	HMI_SL_PB.AckFW.Enable			:= VAR_StatusSafetyScanning = 0		AND VAR_StatusSafetySafeKeyChanged = 0	AND VAR_StatusSafetyNbOfUdId = 0	AND VAR_StatusSafetyNbOfDiffFW > 0	AND VAR_AllowedSafeButton;
	HMI_SL_PB.LedTest.Enable		:= VAR_StatusSafetyScanning = 0		AND VAR_SafeOSState <> 0				AND NOT(VAR_CPUSafetyNotFound)		AND VAR_AllowedSafeButton;
	HMI_SL_PB.Scan.Enable			:= VAR_StatusSafetyScanning = 0		AND VAR_SafeOSState <> 0				AND NOT(VAR_CPUSafetyNotFound)		AND VAR_AllowedSafeButton;

	HMI_SL_PB.Ack_SK.Blink			:= (VAR_StatusSafetyScanning = 0	OR (VAR_StatusSafetyScanning = 1		AND HMI_SL_Info.Led.FAIL = 2		AND HMI_SL_Info.Led.RE <> 0))		AND VAR_StatusSafetySafeKeyChanged = 1	AND VAR_StatusSafetyRemoteControl.Status = 255;
	HMI_SL_PB.Ack1UdId.Blink		:= VAR_StatusSafetyScanning = 0		AND VAR_StatusSafetySafeKeyChanged = 0	AND VAR_StatusSafetyNbOfUdId = 1	AND VAR_StatusSafetyRemoteControl.Status = 255;
	HMI_SL_PB.Ack2UdId.Blink		:= VAR_StatusSafetyScanning = 0		AND VAR_StatusSafetySafeKeyChanged = 0	AND VAR_StatusSafetyNbOfUdId = 2	AND VAR_StatusSafetyRemoteControl.Status = 255;
	HMI_SL_PB.Ack3UdId.Blink		:= VAR_StatusSafetyScanning = 0		AND VAR_StatusSafetySafeKeyChanged = 0	AND VAR_StatusSafetyNbOfUdId = 3	AND VAR_StatusSafetyRemoteControl.Status = 255;
	HMI_SL_PB.Ack4UdId.Blink		:= VAR_StatusSafetyScanning = 0		AND VAR_StatusSafetySafeKeyChanged = 0	AND VAR_StatusSafetyNbOfUdId = 4	AND VAR_StatusSafetyRemoteControl.Status = 255;
	HMI_SL_PB.AckMore4UdId.Blink	:= VAR_StatusSafetyScanning = 0		AND VAR_StatusSafetySafeKeyChanged = 0	AND VAR_StatusSafetyNbOfUdId > 4	AND VAR_StatusSafetyRemoteControl.Status = 255;
	HMI_SL_PB.AckFW.Blink			:= VAR_StatusSafetyScanning = 0		AND VAR_StatusSafetySafeKeyChanged = 0	AND VAR_StatusSafetyNbOfUdId = 0	AND VAR_StatusSafetyNbOfDiffFW > 0	AND VAR_StatusSafetyRemoteControl.Status = 255;

	HMI_SL_PB.Ack_SK.LampON			:= HMI_SL_PB.Ack_SK.ON;
	HMI_SL_PB.Ack1UdId.LampON		:= HMI_SL_PB.Ack1UdId.ON;
	HMI_SL_PB.Ack2UdId.LampON		:= HMI_SL_PB.Ack2UdId.ON;
	HMI_SL_PB.Ack3UdId.LampON		:= HMI_SL_PB.Ack3UdId.ON;
	HMI_SL_PB.Ack4UdId.LampON		:= HMI_SL_PB.Ack4UdId.ON;
	HMI_SL_PB.AckMore4UdId.LampON	:= HMI_SL_PB.AckMore4UdId.ON;
	HMI_SL_PB.AckFW.LampON			:= HMI_SL_PB.AckFW.ON;
	HMI_SL_PB.LedTest.LampON		:= HMI_SL_PB.LedTest.ON;
	HMI_SL_PB.Scan.LampON			:= HMI_SL_PB.Scan.ON;

	VAR_SafeLogicStatus.FailSafe			:= (VAR_StatusSafetyRemoteControl.FailSafe					<> cFAIL_SAFE_OK);
	VAR_SafeLogicStatus.FirmwareAcknowledge	:= (VAR_StatusSafetyRemoteControl.NumberOfDiffFirmware	 	<> 0);
	VAR_SafeLogicStatus.NoExecution			:= (VAR_SafeOSState = cNO_EXECUTION);
	VAR_SafeLogicStatus.RunDebug			:= (VAR_SafeOSState = cRUN_DEBUG);
	VAR_SafeLogicStatus.RunSafe				:= (VAR_SafeOSState = cRUN_SAFE);
	VAR_SafeLogicStatus.SafeKeyExchange		:= (VAR_StatusSafetyRemoteControl.SafeKeyChanged 			<> 0);
	VAR_SafeLogicStatus.Scan				:= (VAR_StatusSafetyRemoteControl.Scanning					<> 0);
	VAR_SafeLogicStatus.ModuleExchange		:= (VAR_StatusSafetyRemoteControl.NumberOfUdIdMismatches	<> 0);
	VAR_SafeLogicStatus.ModuleMissing		:= (VAR_StatusSafetyRemoteControl.NumberOfMissingModules	<> 0);

	HMI_MSG[300]	:= (NOT VAR_SafeLogicStatus.RunSafe AND NOT VAR_SafeLogicStatus.RunDebug) OR VAR_SafeLogicStatus.FailSafe;
	HMI_MSG[301]	:= VAR_SafeLogicStatus.FirmwareAcknowledge OR VAR_SafeLogicStatus.SafeKeyExchange OR (VAR_SafeLogicStatus.ModuleExchange <> 0);
	HMI_MSG[302]	:= VAR_SafeLogicStatus.RunDebug;
END_PROGRAM
```

#### Variables.var - Local variables
```iecst
VAR
	VAR_Index : UINT;
	VAR_Subindex : USINT;
	FB_RemoteEplSDOWrite : EplSDOWrite;
	FB_RemoteEplSDORead : EplSDORead;
	VAR_SafeOSState : UDINT;
	VAR_CPUSafetyNotFound : BOOL;
	TMR_TON_Read : TON;
	CMD_SafetyRemoteControl : CmdRemoteControl_Type;
	VAR_SafeRemoteControl_Step : SafeLogicCtrl_Status;
	VAR_StatusSafetyRemoteControl : StatusRemoteControl_Type;
	VAR_ModuleSafetyMissing : ARRAY[0..100] OF BOOL;
	VAR_AllowedSafeButton : BOOL;
	VAR_SafeAuthor : STRING[32];
	VAR_SafeCRC : UDINT;
	VAR_SafeTime : DATE_AND_TIME;
	VAR_SafeTime_DTStruct : DTStructure;
	i : INT;
	j : INT;
	VAR_NoUpdateStatus : BOOL;
	VAR_Temp : STRING[4];
	VAR_StatusSafetyScanning : USINT;
	VAR_StatusSafetySafeKeyChanged : USINT;
	VAR_StatusSafetyNbOfUdId : UINT;
	VAR_StatusSafetyNbOfDiffFW : UINT;
	VAR_SafetyDeviceAdress : STRING[20];
END_VAR
```

#### Types.typ
```iecst
TYPE
	CmdRemoteControl_Type : 	STRUCT
		Command : UINT;
		Number : UINT;
		Data : UINT;
		Password : ARRAY[0..15]OF USINT;
		NewPassword : ARRAY[0..15]OF USINT;
	END_STRUCT;
	StatusRemoteControl_Type : 	STRUCT
		Command : UINT;
		Number : UINT;
		Status : UINT;
		State : UINT;
		EnterData : UINT;
		EnterNumber : UINT;
		EnterExecuteStatus : UINT;
		SafeOSstate : USINT;
		SafeKeyChanged : USINT;
		LedTestActive : USINT;
		Scanning : USINT;
		OpenSafetyState : USINT;
		FailSafe : USINT;
		NumberOfMissingModules : UINT;
		NumberOfUdIdMismatches : UINT;
		NumberOfDiffFirmware : UINT;
		SAddr : ARRAY[0..100]OF UINT;
		MissingModules : ARRAY[0..15]OF USINT;
		UdIdMismatches : ARRAY[0..15]OF USINT;
		DiffFirmware : ARRAY[0..15]OF USINT;
	END_STRUCT;
	SafeLogicCtrl_Status :
		(
		SafeLogic_Wait := 16#0,
		SafeLogic_ReadOsStatus := 16#5,
		SafeLogic_CMD_ReadStatus := 16#10,
		SafeLogic_ReadStatus := 16#11,
		SafeLogic_ReadCRC := 16#12,
		SafeLogic_ReadTime := 16#13,
		SafeLogic_ReadAuthor := 16#14,
		SafeLogic_CMD_Write := 16#19,
		SafeLogic_AckMore4UdId := 16#20,
		SafeLogic_Ack4UdId := 16#30,
		SafeLogic_Ack3UdId := 16#40,
		SafeLogic_Ack2UdId := 16#50,
		SafeLogic_Ack1UdId := 16#60,
		SafeLogic_Ack_FW := 16#100,
		SafeLogic_Ack_SK := 16#200,
		SafeLogic_LedTest := 16#1000,
		SafeLogic_Scan := 16#2000,
		SafeLogic_SK_Copy := 16#3000,
		SafeLogic_SK_ResumeCopy := 16#4000,
		SafeLogic_SK_ChgPassword := 16#5000,
		SafeLogic_SK_Format := 16#6000
		);
END_TYPE
```

#### Constants.var - Local constants
```iecst
VAR CONSTANT
	cINVALID : USINT := 16#00;
	cON : USINT := 16#0F;
	cLOADING : USINT := 16#33;
	cSTOP_SAFE : USINT := 16#55;
	cRUN_SAFE : USINT := 16#66;
	cHALT_SAFE : USINT := 16#99;
	cSTOP_DEBUG : USINT := 16#AA;
	cRUN_DEBUG : USINT := 16#CC;
	cNO_EXECUTION : USINT := 16#F0;
	cFAIL_SAFE_OK : USINT := 16#55;
	CST_SafePasswordBlank : ARRAY[0..15] OF USINT := [212,29,140,217,143,0,178,4,233,128,9,152,236,248,66,126]; (*Password of the SafeKey coded MD5*)
	CST_SafePasswordNull : ARRAY[0..15] OF USINT := [16(0)]; (*Password of the SafeKey coded MD5*)
END_VAR
```

### Package Logical/12_MAU/1290_Logger - Logger: software change logger 

### Program Logical/12_MAU/1290_Logger/MAU_Logger (IEC) - MAU_Logger Main Program - C#7 - 20.4ms

#### MAU_Logger.st - Cyclic code
```iecst
PROGRAM _CYCLIC
	(* Software object logging *)
	swChg_0.refreshTime 		:= T#1m;
	swChg_0.logLevel			:= arEVENTLOG_SEVERITY_INFO;
	swChg_0.enable				:= TRUE;
	swChg_0();
END_PROGRAM
```

#### Variables.var - Local variables
```iecst
(*****************************************                  MACHINE SYNCHRONIZATION LOGGING             ***************************************************************************************************************)
VAR
	synchLog_0 : SynchLog;
END_VAR
(*****************************************                   UPS LOGGING                                                         ***************************************************************************************************************)
VAR
	upsIO : Sidel_UpsIo_typ;
	upsEvt : LogSupplyEvents;
END_VAR
(*****************************************                   SOFTWARE OBJECT LOGGING                               ***************************************************************************************************************)
VAR
	swChg_0 : SwChg;
	pippo :BOOL;
END_VAR
```

### Package Logical/28_CFG - Machine configuration manager

### Program Logical/28_CFG/CFG (IEC) - CFG Main Program - C#6 200ms

#### Cyclic.sfc - Cyclic code
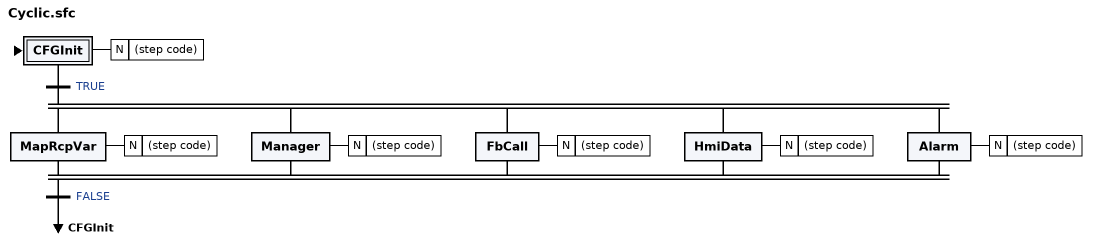
```iecst
PROGRAM _CYCLIC
INITIAL_STEP CFGInit:
CFG_MC;
CFG_Par;
HMI_PAO_2;
CFG_ITC;
CFG_OPS;
END_STEP
TRANSITION FROM CFGInit TO (MapRcpVar,Manager,FbCall,HmiData,Alarm):=
TRUE
END_TRANSITION
STEP MapRcpVar:
pMpLinkRecipeCsv					:= ADR(gRecipeCsv);

(* MpRecipeCsv - Initialization *)
FB_MpRecipeCsv.MpLink				:= pMpLinkRecipeCsv;
FB_MpRecipeCsv.DeviceName			:= ADR(CST_DeviceName);
FB_MpRecipeCsv.FileName				:= ADR(VAR_FileName);
FB_MpRecipeCsv.Header				:= ADR(VAR_Header);
FB_MpRecipeCsv.Enable				:= TRUE;

IF AID.DataOut.ProjectType = CST_AID_ProjectMachine THEN
	(* MpRecipePar - Motion Configuration *)
	FB_MpRecipeRegPar_Motion.MpLink		:= FB_MpRecipeCsv.MpLink;
	FB_MpRecipeRegPar_Motion.Category	:= ADR(VAR_CategoryMotion);
	FB_MpRecipeRegPar_Motion.PVName		:= ADR(VAR_PvNameMotion);
	FB_MpRecipeRegPar_Motion.Enable		:= TRUE;

	(* MpRecipePar - Hmi Pao *)
	FB_MpRecipeRegPar_Hmi.MpLink		:= FB_MpRecipeCsv.MpLink;
	FB_MpRecipeRegPar_Hmi.Category		:= ADR(VAR_CategoryHmi);
	FB_MpRecipeRegPar_Hmi.PVName		:= ADR(VAR_PvNameHmi);
	FB_MpRecipeRegPar_Hmi.Enable		:= TRUE;

	(* MpRecipePar - Operator Safety Configuration *)
	FB_MpRecipeRegPar_CfgOps.MpLink		:= FB_MpRecipeCsv.MpLink;
	FB_MpRecipeRegPar_CfgOps.Category	:= ADR(VAR_CategoryCfgDoor);
	FB_MpRecipeRegPar_CfgOps.PVName		:= ADR(VAR_PvNameCfgDoor);
	FB_MpRecipeRegPar_CfgOps.Enable		:= TRUE;

	(* MpRecipePar - Capper Configuration *)
	FB_MpRecipeRegPar_CfgCap.MpLink		:= FB_MpRecipeCsv.MpLink;
	FB_MpRecipeRegPar_CfgCap.Category	:= ADR(VAR_CategoryCfgCap);
	FB_MpRecipeRegPar_CfgCap.PVName		:= ADR(VAR_PvNameCfgCap);
	FB_MpRecipeRegPar_CfgCap.Enable		:= TRUE;
END_IF

(* MpRecipePar - Machine configuration *)
FB_MpRecipeRegPar_Config.MpLink		:= FB_MpRecipeCsv.MpLink;
FB_MpRecipeRegPar_Config.Category	:= ADR(VAR_CategoryConfig);
FB_MpRecipeRegPar_Config.PVName		:= ADR(VAR_PvNameConfig);
FB_MpRecipeRegPar_Config.Enable		:= TRUE;

(* MpRecipePar - Itc Configuration *)
FB_MpRecipeRegPar_Itc.MpLink		:= FB_MpRecipeCsv.MpLink;
FB_MpRecipeRegPar_Itc.Category		:= ADR(VAR_CategoryItc);
FB_MpRecipeRegPar_Itc.PVName		:= ADR(VAR_PvNameItc);
FB_MpRecipeRegPar_Itc.Enable		:= TRUE;

(* File Manager *)
(* Folder create *)
FB_DirCreate.enable					:= TRUE;
FB_DirCreate.pDevice				:= ADR(CST_RootName);
FB_DirCreate.pName					:= ADR(CST_DirName);
END_STEP
STEP Manager:
CsvManager;
FileManager;
END_STEP
STEP FbCall:
FB_MpRecipeCsv;
FB_MpRecipeRegPar_Motion;
FB_MpRecipeRegPar_Config;
FB_MpRecipeRegPar_CfgCap;
FB_MpRecipeRegPar_Hmi;
FB_MpRecipeRegPar_Itc;
FB_MpRecipeRegPar_CfgOps;
END_STEP
STEP HmiData:
HmiVariablesBrowse;

HMI_PB[PB_CFG_SavePao].Enable		:= VAR_CsvMngState = 800;
HMI_PB[PB_CFG_SavePao].Visibility	:= TRUE;
HMI_PB[PB_CFG_SavePao].LampON		:= HMI_PB[PB_CFG_SavePao].ON;
HMI_PB[PB_CFG_SavePao].Blink		:= VAR_CsvMngState >= 1050 AND VAR_CsvMngState <= 1099 ;

HMI_PB[PB_CFG_LoadPao].Enable		:= VAR_CsvMngState = 800;
HMI_PB[PB_CFG_LoadPao].Visibility	:= TRUE;
HMI_PB[PB_CFG_LoadPao].LampON		:= HMI_PB[PB_CFG_LoadPao].ON;
HMI_PB[PB_CFG_LoadPao].Blink		:= VAR_CsvMngState >= 1000  AND VAR_CsvMngState <= 1049;

HMI_PB[PB_CFG_SaveCfg].Enable		:= VAR_CsvMngState = 800 AND VAR_InitialVariableName <> '';
HMI_PB[PB_CFG_SaveCfg].Visibility	:= TRUE;
HMI_PB[PB_CFG_SaveCfg].LampON		:= HMI_PB[PB_CFG_SaveCfg].ON;
HMI_PB[PB_CFG_SaveCfg].Blink		:= (VAR_CsvMngState >= 1150 AND VAR_CsvMngState <= 1199) OR (VAR_CsvMngState >= 1250 AND VAR_CsvMngState <= 1299);

HMI_PB[PB_CFG_LoadCfg].Enable		:= VAR_CsvMngState = 800 AND VAR_InitialVariableName <> '';
HMI_PB[PB_CFG_LoadCfg].Visibility	:= TRUE;
HMI_PB[PB_CFG_LoadCfg].LampON		:= HMI_PB[PB_CFG_LoadCfg].ON;
HMI_PB[PB_CFG_LoadCfg].Blink		:= (VAR_CsvMngState >= 1100 AND VAR_CsvMngState <= 1149) OR (VAR_CsvMngState >= 1200 AND VAR_CsvMngState <= 1249);
END_STEP
STEP Alarm:
//V4.A.A.1.6.13
ALR[110].Active := CFG.DataOut.CfgDefault OR CFG.DataOut.ItcDefault OR CFG.DataOut.PaoDefault OR CFG.DataOut.CfgCapDefault OR CFG.DataOut.MotionDefault OR CFG.DataOut.OPSDefault;
ALR[111].Active := HMI_MachineId = 'Error Name';
END_STEP
TRANSITION FROM (MapRcpVar,Manager,FbCall,HmiData,Alarm) TO CFGInit:=
FALSE
END_TRANSITION
(* @SFCISJUMP := 'CFGInit' *)
END_PROGRAM
```

#### Constants.var - Local variables
```iecst
VAR CONSTANT
	CST_DeviceName : STRING[16] := 'RECIPE';
	CST_RootName : STRING[16] := 'ROOT';
	CST_DirName : STRING[16] := 'Files';
	CST_DefaultHeader : MpRecipeCsvHeaderType := (Name:='Default Value');
END_VAR
```

#### Variables.var - Local variables
```iecst
VAR
	StFmState : INT;
	VAR_CsvMngState : INT;
	VAR_PV_NinfoState : UINT;
	VAR_FmCmd : FmCmd_Type;
	VAR_FmAck : FmAck_Type;
END_VAR
(*Function Block*)
(*MpRecipe*)
VAR
	FB_MpRecipeCsv : MpRecipeCsv;
	FB_MpRecipeRegPar_Config : MpRecipeRegPar;
	FB_MpRecipeRegPar_Hmi : MpRecipeRegPar;
	FB_MpRecipeRegPar_CfgOps : MpRecipeRegPar;
	FB_MpRecipeRegPar_Itc : MpRecipeRegPar;
	FB_MpRecipeRegPar_Motion : MpRecipeRegPar;
	FB_MpRecipeRegPar_CfgCap : MpRecipeRegPar;
	FB_DirCreate : DirCreate;
	pMpLinkRecipeCsv : UDINT;
END_VAR
(*-----*)
VAR
	VAR_FileName : STRING[14];
	VAR_Header : MpRecipeCsvHeaderType;
	VAR_HmiPaoName : STRING[20];
	VAR_CfgPaoName : STRING[20];
	VAR_CfgDoorName : STRING[20];
	VAR_CfgMotionName : STRING[20];
	VAR_CfgItcName : STRING[20];
	VAR_CfgCapName : STRING[20];
	VAR_CategoryConfig : STRING[50] := 'CFG_Par';
	VAR_PvNameConfig : STRING[100] := 'CFG_Par';
	VAR_CategoryHmi : STRING[50] := 'HMI_PAO_2';
	VAR_PvNameHmi : STRING[100] := 'HMI_PAO_2';
	VAR_CategoryMotion : STRING[50] := 'CFG_MC';
	VAR_PvNameMotion : STRING[100] := 'CFG_MC';
	VAR_CategoryItc : STRING[50] := 'CFG_ITC';
	VAR_PvNameItc : STRING[100] := 'CFG_ITC';
	VAR_CategoryCfgDoor : STRING[50] := 'CFG_OPS';
	VAR_PvNameCfgDoor : STRING[100] := 'CFG_OPS';
	VAR_CategoryCfgCap : STRING[50] := 'CFG_Cap';
	VAR_PvNameCfgCap : STRING[100] := 'CFG_Cap_Par';
	VAR_ItemName : STRING[100];
	VAR_InitialVariableName : STRING[100];
	VAR_VariableName : STRING[100];
	VAR_DType : UDINT;
	VAR_address : UDINT;
	VAR_Dim : UINT;
	VAR_Len : UDINT;
	VAR_DType2 : UDINT;
	VAR_Dim2 : UINT;
	VAR_Len2 : UDINT;
	var_i : UDINT;
	VAR_Level : INT;
	VAR_array : STRING[3];
	VAR_LastElement : INT;
	VAR_LastElementOld : INT;
	VAR_Page : INT;
END_VAR
```

#### Types.typ - Local data types
```iecst
TYPE
	FmCmd_Type : 	STRUCT
		FolderCreate : BOOL;
		Load : BOOL;
		Save : BOOL;
	END_STRUCT;
	FmAck_Type : 	STRUCT
		CommandError : BOOL;
		CommandBusy : BOOL;
		CommandDone : BOOL;
		ErrorCode : UINT;
		ErroreState : FileManagerError_Type;
	END_STRUCT;
	FileManagerError_Type :
		(
		NO_ERROR,
		ERR_FOLDER_CREATE,
		ERR_LOAD,
		ERR_SAVE
		);
END_TYPE
```
